(* PLC project Adressering.ecp, WAGO e!COCKPIT e!COCKPIT *)
(* stored: creationDateTime 2021-01-18T14:20:23.2110188, modificationDateTime 2021-01-18T11:51:27.6823754 *)

TYPE dtRomtype_99999999999999 : STRUCT
  RB601_V : BOOL;  (* Bevegelse *)
  RB602_V : BOOL;  (* Bevegelse *)
  RB603_V : BOOL;  (* Bevegelse *)
  RB604_V : BOOL;  (* Bevegelse *)
  RB605_V : BOOL;  (* Bevegelse *)
  RB606_V : BOOL;  (* Bevegelse *)
  RB607_V : BOOL;  (* Bevegelse *)
  RB608_V : BOOL;  (* Bevegelse *)
  RB609_V : BOOL;  (* Bevegelse *)
  RB601_HVAC : BOOL;  (* HVAC signal *)
  RB602_HVAC : BOOL;  (* HVAC signal *)
  RB603_HVAC : BOOL;  (* HVAC signal *)
  RB604_HVAC : BOOL;  (* HVAC signal *)
  RB605_HVAC : BOOL;  (* HVAC signal *)
  RB606_HVAC : BOOL;  (* HVAC signal *)
  RB607_HVAC : BOOL;  (* HVAC signal *)
  RB608_HVAC : BOOL;  (* HVAC signal *)
  RB609_HVAC : BOOL;  (* HVAC signal *)
  RT601_CT : REAL;  (* Rom temperatur *)
  RT602_CT : REAL;  (* Rom temperatur *)
  RT602_SP : REAL;  (* Temperatur SP *)
  RT603_CT : REAL;  (* Rom temperatur *)
  RT603_SP : REAL;  (* Temperatur SP *)
  RT604_CT : REAL;  (* Rom temperatur *)
  RT604_SP : REAL;  (* Temperatur SP *)
  RT605_CT : REAL;  (* Rom temperatur *)
  RT605_SP : REAL;  (* Temperatur SP *)
  RT606_CT : REAL;  (* Rom temperatur *)
  RT606_SP : REAL;  (* Temperatur SP *)
  RT607_CT : REAL;  (* Rom temperatur *)
  RT607_SP : REAL;  (* Temperatur SP *)
  RT608_CT : REAL;  (* Rom temperatur *)
  RT608_SP : REAL;  (* Temperatur SP *)
  RT609_CT : REAL;  (* Rom temperatur *)
  RT609_SP : REAL;  (* Temperatur SP *)
  RT601_SP_D : REAL;  (* Temperatur SP *)
  RT601_SP_S : REAL;  (* Temperatur SP standby *)
  RT601_SP_N : REAL;  (* Temperatur SP nattsenk *)
  RT601_SP_F : REAL;  (* Temperatur SP frostsikring *)
  RT601_CS : REAL;  (* Aktivt temperatur SP *)
  OPM : INT;  (* Rom modus *)
  OPM_CV : INT;  (* Rom modus verdi *)
  RY601_CV : REAL;  (* Co2 Nivaa *)
  RY602_CV : REAL;  (* Co2 Nivaa *)
  RY603_CV : REAL;  (* Co2 Nivaa *)
  RY604_CV : REAL;  (* Co2 Nivaa *)
  RY605_CV : REAL;  (* Co2 Nivaa *)
  RY606_CV : REAL;  (* Co2 Nivaa *)
  RY607_CV : REAL;  (* Co2 Nivaa *)
  RY608_CV : REAL;  (* Co2 Nivaa *)
  RY609_CV : REAL;  (* Co2 Nivaa *)
  RY601_SP : REAL;  (* Co2 SP *)
  RY601_OP : REAL;  (* Co2 paadrag *)
  LH601_OP : REAL;  (* Varmepaadrag *)
  LH602_OP : REAL;  (* Varmepaadrag *)
  LH603_OP : REAL;  (* Varmepaadrag *)
  LH604_OP : REAL;  (* Varmepaadrag *)
  LH605_OP : REAL;  (* Varmepaadrag *)
  LH606_OP : REAL;  (* Varmepaadrag *)
  LH607_OP : REAL;  (* Varmepaadrag *)
  LH608_OP : REAL;  (* Varmepaadrag *)
  LH609_OP : REAL;  (* Varmepaadrag *)
  LH601_MAN : BOOL;  (* Force LH *)
  LH601_CMD : BOOL;  (* LH601_CMD *)
  LH602_CMD : BOOL;  (* LH602_CMD *)
  LH603_CMD : BOOL;  (* LH603_CMD *)
  LH604_CMD : BOOL;  (* LH604_CMD *)
  LH605_CMD : BOOL;  (* LH605_CMD *)
  LH606_CMD : BOOL;  (* LH606_CMD *)
  LH607_CMD : BOOL;  (* LH607_CMD *)
  LH608_CMD : BOOL;  (* LH608_CMD *)
  LH609_CMD : BOOL;  (* LH609_CMD *)
  LC601_OP : REAL;  (* LC601_OP *)
  LC602_OP : REAL;  (* LC602_OP *)
  LC603_OP : REAL;  (* LC603_OP *)
  LC604_OP : REAL;  (* LC604_OP *)
  LC605_OP : REAL;  (* LC605_OP *)
  LC606_OP : REAL;  (* LC606_OP *)
  LC607_OP : REAL;  (* LC607_OP *)
  LC608_OP : REAL;  (* LC608_OP *)
  LC609_OP : REAL;  (* LC609_OP *)
  LC601_MAN : BOOL;  (* Force LC *)
  LC601_CMD : BOOL;  (* LC601_CMD *)
  LC602_CMD : BOOL;  (* LC602_CMD *)
  LC603_CMD : BOOL;  (* LC603_CMD *)
  LC604_CMD : BOOL;  (* LC604_CMD *)
  LC605_CMD : BOOL;  (* LC605_CMD *)
  LC606_CMD : BOOL;  (* LC606_CMD *)
  LC607_CMD : BOOL;  (* LC607_CMD *)
  LC608_CMD : BOOL;  (* LC608_CMD *)
  LC609_CMD : BOOL;  (* LC609_CMD *)
  RT601_SP : REAL;  (* Temperatur SP feedback *)
  RT601_SP_FB : REAL;  (* Temperatur SP *)
  RT601_SP_IN : REAL;  (* Temperatur SP lokalt panel *)
  RT602_SP_FB : REAL;  (* Temperatur SP *)
  RT602_SP_IN : REAL;  (* Temperatur SP lokalt panel *)
  RT603_SP_FB : REAL;  (* Temperatur SP *)
  RT603_SP_IN : REAL;  (* Temperatur SP lokalt panel *)
  RT604_SP_FB : REAL;  (* Temperatur SP *)
  RT604_SP_IN : REAL;  (* Temperatur SP lokalt panel *)
  RT605_SP_FB : REAL;  (* Temperatur SP *)
  RT605_SP_IN : REAL;  (* Temperatur SP lokalt panel *)
  RT606_SP_FB : REAL;  (* Temperatur SP *)
  RT606_SP_IN : REAL;  (* Temperatur SP lokalt panel *)
  RT607_SP_FB : REAL;  (* Temperatur SP *)
  RT607_SP_IN : REAL;  (* Temperatur SP lokalt panel *)
  RT608_SP_FB : REAL;  (* Temperatur SP *)
  RT608_SP_IN : REAL;  (* Temperatur SP lokalt panel *)
  RT609_SP_FB : REAL;  (* Temperatur SP *)
  RT609_SP_IN : REAL;  (* Temperatur SP lokalt panel *)
  LU601_V : BOOL;  (* Befukter status *)
  LU602_V : BOOL;  (* Befukter status *)
  LU603_V : BOOL;  (* Befukter status *)
  LU604_V : BOOL;  (* Befukter status *)
  LU605_V : BOOL;  (* Befukter status *)
  LU606_V : BOOL;  (* Befukter status *)
  LU607_V : BOOL;  (* Befukter status *)
  LU608_V : BOOL;  (* Befukter status *)
  LU609_V : BOOL;  (* Befukter status *)
  LU601_AL : BOOL;  (* Befukter alarm/feil *)
  LU602_AL : BOOL;  (* Befukter alarm/feil *)
  LU603_AL : BOOL;  (* Befukter alarm/feil *)
  LU604_AL : BOOL;  (* Befukter alarm/feil *)
  LU605_AL : BOOL;  (* Befukter alarm/feil *)
  LU606_AL : BOOL;  (* Befukter alarm/feil *)
  LU607_AL : BOOL;  (* Befukter alarm/feil *)
  LU608_AL : BOOL;  (* Befukter alarm/feil *)
  LU609_AL : BOOL;  (* Befukter alarm/feil *)
  LU601_CMD : BOOL;  (* Befukter tillat start *)
  LU602_CMD : BOOL;  (* Befukter tillat start *)
  LU603_CMD : BOOL;  (* Befukter tillat start *)
  LU604_CMD : BOOL;  (* Befukter tillat start *)
  LU605_CMD : BOOL;  (* Befukter tillat start *)
  LU606_CMD : BOOL;  (* Befukter tillat start *)
  LU607_CMD : BOOL;  (* Befukter tillat start *)
  LU608_CMD : BOOL;  (* Befukter tillat start *)
  LU609_CMD : BOOL;  (* Befukter tillat start *)
END_STRUCT;
END_TYPE

TYPE dtRomtype_2210111100111 : STRUCT
  RB601_V : BOOL;  (* Bevegelse *)
  RB602_V : BOOL;  (* Bevegelse *)
  RB601_HVAC : BOOL;  (* HVAC signal *)
  RB602_HVAC : BOOL;  (* HVAC signal *)
  RT601_CT : REAL;  (* Rom temperatur *)
  RT601_SP_D : REAL;  (* Temperatur SP *)
  RT601_SP_S : REAL;  (* Temperatur SP standby *)
  RT601_SP_N : REAL;  (* Temperatur SP nattsenk *)
  RT601_SP_F : REAL;  (* Temperatur SP frostsikring *)
  RT601_CS : REAL;  (* Aktivt temperatur SP *)
  OPM : INT;  (* Rom modus *)
  OPM_CV : INT;  (* Rom modus verdi *)
  LH601_OP : REAL;  (* Varmepaadrag *)
  LH601_MAN : BOOL;  (* Force LH *)
  LH601_CMD : BOOL;  (* LH601_CMD *)
  LC601_OP : REAL;  (* LC601_OP *)
  LC601_MAN : BOOL;  (* Force LC *)
  LC601_CMD : BOOL;  (* LC601_CMD *)
  LU601_V : BOOL;  (* Befukter status *)
  LU601_AL : BOOL;  (* Befukter alarm/feil *)
  LU601_CMD : BOOL;  (* Befukter tillat start *)
END_STRUCT;
END_TYPE

TYPE dtRomtype_1120011 : STRUCT
  RB601_V : BOOL;  (* Bevegelse *)
  RB601_HVAC : BOOL;  (* HVAC signal *)
  RT601_CT : REAL;  (* Rom temperatur *)
  RT602_CT : REAL;  (* Rom temperatur *)
  RT602_SP : REAL;  (* Temperatur SP *)
  RT601_SP_D : REAL;  (* Temperatur SP *)
  RT601_SP_S : REAL;  (* Temperatur SP standby *)
  RT601_SP_N : REAL;  (* Temperatur SP nattsenk *)
  RT601_SP_F : REAL;  (* Temperatur SP frostsikring *)
  RT601_CS : REAL;  (* Aktivt temperatur SP *)
  OPM : INT;  (* Rom modus *)
  OPM_CV : INT;  (* Rom modus verdi *)
  LH601_CMD : BOOL;  (* LH601_CMD *)
  LH601_MAN : BOOL;  (* Force LH *)
  LC601_OP : REAL;  (* LC601_OP *)
  LC601_MAN : BOOL;  (* Force LC *)
END_STRUCT;
END_TYPE

TYPE dtRomtype_11 : STRUCT
  RB601_V : BOOL;  (* Bevegelse *)
  RB601_HVAC : BOOL;  (* HVAC signal *)
END_STRUCT;
END_TYPE

TYPE dtRomtype_1121 : STRUCT
  RB601_V : BOOL;  (* Bevegelse *)
  RB601_HVAC : BOOL;  (* HVAC signal *)
  RT601_CT : REAL;  (* Rom temperatur *)
  RT602_CT : REAL;  (* Rom temperatur *)
  RT602_SP : REAL;  (* Temperatur SP *)
  RT601_SP_D : REAL;  (* Temperatur SP *)
  RT601_SP_S : REAL;  (* Temperatur SP standby *)
  RT601_SP_N : REAL;  (* Temperatur SP nattsenk *)
  RT601_SP_F : REAL;  (* Temperatur SP frostsikring *)
  RT601_CS : REAL;  (* Aktivt temperatur SP *)
  OPM : INT;  (* Rom modus *)
  OPM_CV : INT;  (* Rom modus verdi *)
  RY601_CV : REAL;  (* Co2 Nivaa *)
  RY601_SP : REAL;  (* Co2 SP *)
  RY601_OP : REAL;  (* Co2 paadrag *)
END_STRUCT;
END_TYPE

TYPE dtRomtype_112001 : STRUCT
  RB601_V : BOOL;  (* Bevegelse *)
  RB601_HVAC : BOOL;  (* HVAC signal *)
  RT601_CT : REAL;  (* Rom temperatur *)
  RT602_CT : REAL;  (* Rom temperatur *)
  RT602_SP : REAL;  (* Temperatur SP *)
  RT601_SP_D : REAL;  (* Temperatur SP *)
  RT601_SP_S : REAL;  (* Temperatur SP standby *)
  RT601_SP_N : REAL;  (* Temperatur SP nattsenk *)
  RT601_SP_F : REAL;  (* Temperatur SP frostsikring *)
  RT601_CS : REAL;  (* Aktivt temperatur SP *)
  OPM : INT;  (* Rom modus *)
  OPM_CV : INT;  (* Rom modus verdi *)
  LH601_CMD : BOOL;  (* LH601_CMD *)
  LH601_MAN : BOOL;  (* Force LH *)
END_STRUCT;
END_TYPE

TYPE dtRomtype_111 : STRUCT
  RB601_V : BOOL;  (* Bevegelse *)
  RB601_HVAC : BOOL;  (* HVAC signal *)
  RT601_CT : REAL;  (* Rom temperatur *)
  RT601_SP_D : REAL;  (* Temperatur SP *)
  RT601_SP_S : REAL;  (* Temperatur SP standby *)
  RT601_SP_N : REAL;  (* Temperatur SP nattsenk *)
  RT601_SP_F : REAL;  (* Temperatur SP frostsikring *)
  RT601_CS : REAL;  (* Aktivt temperatur SP *)
  OPM : INT;  (* Rom modus *)
  OPM_CV : INT;  (* Rom modus verdi *)
END_STRUCT;
END_TYPE

TYPE dtRomtype_22 : STRUCT
  RB601_V : BOOL;  (* Bevegelse *)
  RB602_V : BOOL;  (* Bevegelse *)
  RB601_HVAC : BOOL;  (* HVAC signal *)
  RB602_HVAC : BOOL;  (* HVAC signal *)
END_STRUCT;
END_TYPE

TYPE dtRomtype_4421011 : STRUCT
  RB601_V : BOOL;  (* Bevegelse *)
  RB602_V : BOOL;  (* Bevegelse *)
  RB603_V : BOOL;  (* Bevegelse *)
  RB604_V : BOOL;  (* Bevegelse *)
  RB601_HVAC : BOOL;  (* HVAC signal *)
  RB602_HVAC : BOOL;  (* HVAC signal *)
  RB603_HVAC : BOOL;  (* HVAC signal *)
  RB604_HVAC : BOOL;  (* HVAC signal *)
  RT601_CT : REAL;  (* Rom temperatur *)
  RT602_CT : REAL;  (* Rom temperatur *)
  RT602_SP : REAL;  (* Temperatur SP *)
  RT601_SP_D : REAL;  (* Temperatur SP *)
  RT601_SP_S : REAL;  (* Temperatur SP standby *)
  RT601_SP_N : REAL;  (* Temperatur SP nattsenk *)
  RT601_SP_F : REAL;  (* Temperatur SP frostsikring *)
  RT601_CS : REAL;  (* Aktivt temperatur SP *)
  OPM : INT;  (* Rom modus *)
  OPM_CV : INT;  (* Rom modus verdi *)
  RY601_CV : REAL;  (* Co2 Nivaa *)
  RY601_SP : REAL;  (* Co2 SP *)
  RY601_OP : REAL;  (* Co2 paadrag *)
  LH601_CMD : BOOL;  (* LH601_CMD *)
  LH601_MAN : BOOL;  (* Force LH *)
  LC601_OP : REAL;  (* LC601_OP *)
  LC601_MAN : BOOL;  (* Force LC *)
END_STRUCT;
END_TYPE

TYPE dtRomtype_003 : STRUCT
  RT601_CT : REAL;  (* Rom temperatur *)
  RT602_CT : REAL;  (* Rom temperatur *)
  RT602_SP : REAL;  (* Temperatur SP *)
  RT603_CT : REAL;  (* Rom temperatur *)
  RT603_SP : REAL;  (* Temperatur SP *)
  RT601_SP_D : REAL;  (* Temperatur SP *)
  RT601_SP_S : REAL;  (* Temperatur SP standby *)
  RT601_SP_N : REAL;  (* Temperatur SP nattsenk *)
  RT601_SP_F : REAL;  (* Temperatur SP frostsikring *)
  RT601_CS : REAL;  (* Aktivt temperatur SP *)
  OPM : INT;  (* Rom modus *)
  OPM_CV : INT;  (* Rom modus verdi *)
END_STRUCT;
END_TYPE

TYPE dtRomtype_1121011 : STRUCT
  RB601_V : BOOL;  (* Bevegelse *)
  RB601_HVAC : BOOL;  (* HVAC signal *)
  RT601_CT : REAL;  (* Rom temperatur *)
  RT602_CT : REAL;  (* Rom temperatur *)
  RT602_SP : REAL;  (* Temperatur SP *)
  RT601_SP_D : REAL;  (* Temperatur SP *)
  RT601_SP_S : REAL;  (* Temperatur SP standby *)
  RT601_SP_N : REAL;  (* Temperatur SP nattsenk *)
  RT601_SP_F : REAL;  (* Temperatur SP frostsikring *)
  RT601_CS : REAL;  (* Aktivt temperatur SP *)
  OPM : INT;  (* Rom modus *)
  OPM_CV : INT;  (* Rom modus verdi *)
  RY601_CV : REAL;  (* Co2 Nivaa *)
  RY601_SP : REAL;  (* Co2 SP *)
  RY601_OP : REAL;  (* Co2 paadrag *)
  LH601_CMD : BOOL;  (* LH601_CMD *)
  LH601_MAN : BOOL;  (* Force LH *)
  LC601_OP : REAL;  (* LC601_OP *)
  LC601_MAN : BOOL;  (* Force LC *)
END_STRUCT;
END_TYPE

TYPE dtRomtype_112 : STRUCT
  RB601_V : BOOL;  (* Bevegelse *)
  RB601_HVAC : BOOL;  (* HVAC signal *)
  RT601_CT : REAL;  (* Rom temperatur *)
  RT602_CT : REAL;  (* Rom temperatur *)
  RT602_SP : REAL;  (* Temperatur SP *)
  RT601_SP_D : REAL;  (* Temperatur SP *)
  RT601_SP_S : REAL;  (* Temperatur SP standby *)
  RT601_SP_N : REAL;  (* Temperatur SP nattsenk *)
  RT601_SP_F : REAL;  (* Temperatur SP frostsikring *)
  RT601_CS : REAL;  (* Aktivt temperatur SP *)
  OPM : INT;  (* Rom modus *)
  OPM_CV : INT;  (* Rom modus verdi *)
END_STRUCT;
END_TYPE

{attribute 'qualified_only'}
VAR_GLOBAL  (* STLV59_563 *)
  STLV59_A_563_KNX_Card_1_Status : BOOL;  (* KNX kort 1 status *)
  STLV59_A_563_000 : dtRomtype_99999999999999;
  STLV59_A_563_001 : dtRomtype_2210111100111;
  STLV59_A_563_002 : dtRomtype_1120011;
  STLV59_A_563_003 : dtRomtype_11;
  STLV59_A_563_004 : dtRomtype_1121;
  STLV59_A_563_005 : dtRomtype_112001;
  STLV59_A_563_006 : dtRomtype_111;
  STLV59_A_563_007 : dtRomtype_112001;
  STLV59_A_563_008 : dtRomtype_112001;
  STLV59_A_563_009 : dtRomtype_112001;
  STLV59_A_563_010 : dtRomtype_112001;
  STLV59_A_563_011 : dtRomtype_112001;
  STLV59_A_563_012 : dtRomtype_112001;
  STLV59_A_563_013 : dtRomtype_112001;
  STLV59_A_563_014 : dtRomtype_22;
  STLV59_A_563_015 : dtRomtype_11;
  STLV59_A_563_016 : dtRomtype_11;
  STLV59_A_563_017 : dtRomtype_112001;
  STLV59_A_563_101 : dtRomtype_112001;
  STLV59_A_563_102 : dtRomtype_112001;
  STLV59_A_563_103 : dtRomtype_4421011;
  STLV59_A_563_109 : dtRomtype_112001;
  STLV59_A_563_201 : dtRomtype_003;
  STLV59_A_563_212 : dtRomtype_1121011;
  STLV59_A_563_213 : dtRomtype_112;
  STLV59_A_563_T2_1 : dtRomtype_112001;
  STLV59_A_563_T2_2 : dtRomtype_112001;
END_VAR

FUNCTION_BLOCK fbRomtype_99999999999999
  VAR_INPUT
    RB601_HVAC : BOOL;
    RB602_HVAC : BOOL;
    RB603_HVAC : BOOL;
    RB604_HVAC : BOOL;
    RB605_HVAC : BOOL;
    RB606_HVAC : BOOL;
    RB607_HVAC : BOOL;
    RB608_HVAC : BOOL;
    RB609_HVAC : BOOL;
    RT601_CT : REAL;
    RT602_CT : REAL;
    RT602_SP : REAL;
    RT603_CT : REAL;
    RT603_SP : REAL;
    RT604_CT : REAL;
    RT604_SP : REAL;
    RT605_CT : REAL;
    RT605_SP : REAL;
    RT606_CT : REAL;
    RT606_SP : REAL;
    RT607_CT : REAL;
    RT607_SP : REAL;
    RT608_CT : REAL;
    RT608_SP : REAL;
    RT609_CT : REAL;
    RT609_SP : REAL;
    RT601_SP_D : REAL;
    RT601_SP_S : REAL;
    RT601_SP_N : REAL;
    RT601_SP_F : REAL;
    OPM : INT;
    RY601_CV : REAL;
    RY602_CV : REAL;
    RY603_CV : REAL;
    RY604_CV : REAL;
    RY605_CV : REAL;
    RY606_CV : REAL;
    RY607_CV : REAL;
    RY608_CV : REAL;
    RY609_CV : REAL;
    RY601_SP : REAL;
    LH601_MAN : BOOL;
    LC601_MAN : BOOL;
    RT601_SP_IN : REAL;
    RT602_SP_IN : REAL;
    RT603_SP_IN : REAL;
    RT604_SP_IN : REAL;
    RT605_SP_IN : REAL;
    RT606_SP_IN : REAL;
    RT607_SP_IN : REAL;
    RT608_SP_IN : REAL;
    RT609_SP_IN : REAL;
    LU601_V : BOOL;
    LU602_V : BOOL;
    LU603_V : BOOL;
    LU604_V : BOOL;
    LU605_V : BOOL;
    LU606_V : BOOL;
    LU607_V : BOOL;
    LU608_V : BOOL;
    LU609_V : BOOL;
    LU601_AL : BOOL;
    LU602_AL : BOOL;
    LU603_AL : BOOL;
    LU604_AL : BOOL;
    LU605_AL : BOOL;
    LU606_AL : BOOL;
    LU607_AL : BOOL;
    LU608_AL : BOOL;
    LU609_AL : BOOL;
  END_VAR
  VAR_OUTPUT
    OPM_CV : INT;
    RT601_CS : REAL;
    RT602_CS : REAL;
    RT603_CS : REAL;
    RT604_CS : REAL;
    RT605_CS : REAL;
    RT606_CS : REAL;
    RT607_CS : REAL;
    RT608_CS : REAL;
    RT609_CS : REAL;
    RY601_OP : REAL;
    LH601_OP : REAL;
    LH602_OP : REAL;
    LH603_OP : REAL;
    LH604_OP : REAL;
    LH605_OP : REAL;
    LH606_OP : REAL;
    LH607_OP : REAL;
    LH608_OP : REAL;
    LH609_OP : REAL;
    LH601_CMD : BOOL;
    LH602_CMD : BOOL;
    LH603_CMD : BOOL;
    LH604_CMD : BOOL;
    LH605_CMD : BOOL;
    LH606_CMD : BOOL;
    LH607_CMD : BOOL;
    LH608_CMD : BOOL;
    LH609_CMD : BOOL;
    LC601_OP : REAL;
    LC602_OP : REAL;
    LC603_OP : REAL;
    LC604_OP : REAL;
    LC605_OP : REAL;
    LC606_OP : REAL;
    LC607_OP : REAL;
    LC608_OP : REAL;
    LC609_OP : REAL;
    LC601_CMD : BOOL;
    LC602_CMD : BOOL;
    LC603_CMD : BOOL;
    LC604_CMD : BOOL;
    LC605_CMD : BOOL;
    LC606_CMD : BOOL;
    LC607_CMD : BOOL;
    LC608_CMD : BOOL;
    LC609_CMD : BOOL;
    LU601_CMD : BOOL;
    LU602_CMD : BOOL;
    LU603_CMD : BOOL;
    LU604_CMD : BOOL;
    LU605_CMD : BOOL;
    LU606_CMD : BOOL;
    LU607_CMD : BOOL;
    LU608_CMD : BOOL;
    LU609_CMD : BOOL;
  END_VAR

(* CFC diagram, written out as Structured Text *)
END_FUNCTION_BLOCK

FUNCTION_BLOCK fbRomtype_2210111100111
  VAR_INPUT
    RB601_HVAC : BOOL;
    RB602_HVAC : BOOL;
    RT601_CT : REAL;
    RT601_SP_D : REAL;
    RT601_SP_S : REAL;
    RT601_SP_N : REAL;
    RT601_SP_F : REAL;
    OPM : INT;
    LH601_MAN : BOOL;
    LC601_MAN : BOOL;
    LU601_V : BOOL;
    LU601_AL : BOOL;
  END_VAR
  VAR_OUTPUT
    OPM_CV : INT;
    RT601_CS : REAL;
    LH601_OP : REAL;
    LH601_CMD : BOOL;
    LC601_OP : REAL;
    LC601_CMD : BOOL;
    LU601_CMD : BOOL;
  END_VAR

(* CFC diagram, written out as Structured Text *)
END_FUNCTION_BLOCK

FUNCTION_BLOCK fbRomtype_1120011
  VAR_INPUT
    RB601_HVAC : BOOL;
    RT601_CT : REAL;
    RT602_CT : REAL;
    RT602_SP : REAL;
    RT601_SP_D : REAL;
    RT601_SP_S : REAL;
    RT601_SP_N : REAL;
    RT601_SP_F : REAL;
    OPM : INT;
    LH601_MAN : BOOL;
    LC601_MAN : BOOL;
  END_VAR
  VAR_OUTPUT
    OPM_CV : INT;
    RT601_CS : REAL;
    RT602_CS : REAL;
    LH601_CMD : BOOL;
    LC601_OP : REAL;
  END_VAR

(* CFC diagram, written out as Structured Text *)
END_FUNCTION_BLOCK

FUNCTION_BLOCK fbRomtype_1121
  VAR_INPUT
    RB601_HVAC : BOOL;
    RT601_CT : REAL;
    RT602_CT : REAL;
    RT602_SP : REAL;
    RT601_SP_D : REAL;
    RT601_SP_S : REAL;
    RT601_SP_N : REAL;
    RT601_SP_F : REAL;
    OPM : INT;
    RY601_CV : REAL;
    RY601_SP : REAL;
  END_VAR
  VAR_OUTPUT
    OPM_CV : INT;
    RT601_CS : REAL;
    RT602_CS : REAL;
    RY601_OP : REAL;
  END_VAR

(* CFC diagram, written out as Structured Text *)
END_FUNCTION_BLOCK

FUNCTION_BLOCK fbRomtype_112001
  VAR_INPUT
    RB601_HVAC : BOOL;
    RT601_CT : REAL;
    RT602_CT : REAL;
    RT602_SP : REAL;
    RT601_SP_D : REAL;
    RT601_SP_S : REAL;
    RT601_SP_N : REAL;
    RT601_SP_F : REAL;
    OPM : INT;
    LH601_MAN : BOOL;
  END_VAR
  VAR_OUTPUT
    OPM_CV : INT;
    RT601_CS : REAL;
    RT602_CS : REAL;
    LH601_CMD : BOOL;
  END_VAR

(* CFC diagram, written out as Structured Text *)
END_FUNCTION_BLOCK

FUNCTION_BLOCK fbRomtype_4421011
  VAR_INPUT
    RB601_HVAC : BOOL;
    RB602_HVAC : BOOL;
    RB603_HVAC : BOOL;
    RB604_HVAC : BOOL;
    RT601_CT : REAL;
    RT602_CT : REAL;
    RT602_SP : REAL;
    RT601_SP_D : REAL;
    RT601_SP_S : REAL;
    RT601_SP_N : REAL;
    RT601_SP_F : REAL;
    OPM : INT;
    RY601_CV : REAL;
    RY601_SP : REAL;
    LH601_MAN : BOOL;
    LC601_MAN : BOOL;
  END_VAR
  VAR_OUTPUT
    OPM_CV : INT;
    RT601_CS : REAL;
    RT602_CS : REAL;
    RY601_OP : REAL;
    LH601_CMD : BOOL;
    LC601_OP : REAL;
  END_VAR

(* CFC diagram, written out as Structured Text *)
END_FUNCTION_BLOCK

FUNCTION_BLOCK fbRomtype_1121011
  VAR_INPUT
    RB601_HVAC : BOOL;
    RT601_CT : REAL;
    RT602_CT : REAL;
    RT602_SP : REAL;
    RT601_SP_D : REAL;
    RT601_SP_S : REAL;
    RT601_SP_N : REAL;
    RT601_SP_F : REAL;
    OPM : INT;
    RY601_CV : REAL;
    RY601_SP : REAL;
    LH601_MAN : BOOL;
    LC601_MAN : BOOL;
  END_VAR
  VAR_OUTPUT
    OPM_CV : INT;
    RT601_CS : REAL;
    RT602_CS : REAL;
    RY601_OP : REAL;
    LH601_CMD : BOOL;
    LC601_OP : REAL;
  END_VAR

(* CFC diagram, written out as Structured Text *)
END_FUNCTION_BLOCK

PROGRAM PRG_563_KNX_1
  VAR
    i : INT := 0;  (* Felles *)
    Interval : OSCAT_BASIC.CLK_PRG;
    typDPT : typDPT;
    KNX_master_1 : WagoAppKNX.FbKNX_Master;  (* Master *)
    M1_001_000_RB601_V : fbDPT_Switch_pro;  (* 000 *)
    M1_002_000_RB602_V : fbDPT_Switch_pro;
    M1_003_000_RB603_V : fbDPT_Switch_pro;
    M1_004_000_RB604_V : fbDPT_Switch_pro;
    M1_005_000_RB605_V : fbDPT_Switch_pro;
    M1_006_000_RB606_V : fbDPT_Switch_pro;
    M1_007_000_RB607_V : fbDPT_Switch_pro;
    M1_008_000_RB608_V : fbDPT_Switch_pro;
    M1_009_000_RB609_V : fbDPT_Switch_pro;
    M1_010_000_RB601_HVAC : fbDPT_Switch_pro;
    M1_011_000_RB602_HVAC : fbDPT_Switch_pro;
    M1_012_000_RB603_HVAC : fbDPT_Switch_pro;
    M1_013_000_RB604_HVAC : fbDPT_Switch_pro;
    M1_014_000_RB605_HVAC : fbDPT_Switch_pro;
    M1_015_000_RB606_HVAC : fbDPT_Switch_pro;
    M1_016_000_RB607_HVAC : fbDPT_Switch_pro;
    M1_017_000_RB608_HVAC : fbDPT_Switch_pro;
    M1_018_000_RB609_HVAC : fbDPT_Switch_pro;
    M1_019_000_RT601_CT : fbDPT_Value_Temp_pro;
    M1_020_000_RT602_CT : fbDPT_Value_Temp_pro;
    M1_021_000_RT603_CT : fbDPT_Value_Temp_pro;
    M1_022_000_RT604_CT : fbDPT_Value_Temp_pro;
    M1_023_000_RT605_CT : fbDPT_Value_Temp_pro;
    M1_024_000_RT606_CT : fbDPT_Value_Temp_pro;
    M1_025_000_RT607_CT : fbDPT_Value_Temp_pro;
    M1_026_000_RT608_CT : fbDPT_Value_Temp_pro;
    M1_027_000_RT609_CT : fbDPT_Value_Temp_pro;
    M1_028_000_RY601_CV : fbDPT_Value_AirQuality_pro;
    M1_029_000_RY602_CV : fbDPT_Value_AirQuality_pro;
    M1_030_000_RY603_CV : fbDPT_Value_AirQuality_pro;
    M1_031_000_RY604_CV : fbDPT_Value_AirQuality_pro;
    M1_032_000_RY605_CV : fbDPT_Value_AirQuality_pro;
    M1_033_000_RY606_CV : fbDPT_Value_AirQuality_pro;
    M1_034_000_RY607_CV : fbDPT_Value_AirQuality_pro;
    M1_035_000_RY608_CV : fbDPT_Value_AirQuality_pro;
    M1_036_000_RY609_CV : fbDPT_Value_AirQuality_pro;
    M1_037_000_LH601_OP : fbDPT_Scaling_pro;
    M1_038_000_LH602_OP : fbDPT_Scaling_pro;
    M1_039_000_LH603_OP : fbDPT_Scaling_pro;
    M1_040_000_LH604_OP : fbDPT_Scaling_pro;
    M1_041_000_LH605_OP : fbDPT_Scaling_pro;
    M1_042_000_LH606_OP : fbDPT_Scaling_pro;
    M1_043_000_LH607_OP : fbDPT_Scaling_pro;
    M1_044_000_LH608_OP : fbDPT_Scaling_pro;
    M1_045_000_LH609_OP : fbDPT_Scaling_pro;
    M1_046_000_LH601_CMD : fbDPT_Switch_pro;
    M1_047_000_LH602_CMD : fbDPT_Switch_pro;
    M1_048_000_LH603_CMD : fbDPT_Switch_pro;
    M1_049_000_LH604_CMD : fbDPT_Switch_pro;
    M1_050_000_LH605_CMD : fbDPT_Switch_pro;
    M1_051_000_LH606_CMD : fbDPT_Switch_pro;
    M1_052_000_LH607_CMD : fbDPT_Switch_pro;
    M1_053_000_LH608_CMD : fbDPT_Switch_pro;
    M1_054_000_LH609_CMD : fbDPT_Switch_pro;
    M1_055_000_LC601_OP : fbDPT_Scaling_pro;
    M1_056_000_LC602_OP : fbDPT_Scaling_pro;
    M1_057_000_LC603_OP : fbDPT_Scaling_pro;
    M1_058_000_LC604_OP : fbDPT_Scaling_pro;
    M1_059_000_LC605_OP : fbDPT_Scaling_pro;
    M1_060_000_LC606_OP : fbDPT_Scaling_pro;
    M1_061_000_LC607_OP : fbDPT_Scaling_pro;
    M1_062_000_LC608_OP : fbDPT_Scaling_pro;
    M1_063_000_LC609_OP : fbDPT_Scaling_pro;
    M1_064_000_LC601_CMD : fbDPT_Switch_pro;
    M1_065_000_LC602_CMD : fbDPT_Switch_pro;
    M1_066_000_LC603_CMD : fbDPT_Switch_pro;
    M1_067_000_LC604_CMD : fbDPT_Switch_pro;
    M1_068_000_LC605_CMD : fbDPT_Switch_pro;
    M1_069_000_LC606_CMD : fbDPT_Switch_pro;
    M1_070_000_LC607_CMD : fbDPT_Switch_pro;
    M1_071_000_LC608_CMD : fbDPT_Switch_pro;
    M1_072_000_LC609_CMD : fbDPT_Switch_pro;
    M1_073_000_RT601_SP : fbDPT_Value_Temp_pro;
    M1_074_000_RT602_SP : fbDPT_Value_Temp_pro;
    M1_075_000_RT603_SP : fbDPT_Value_Temp_pro;
    M1_076_000_RT604_SP : fbDPT_Value_Temp_pro;
    M1_077_000_RT605_SP : fbDPT_Value_Temp_pro;
    M1_078_000_RT606_SP : fbDPT_Value_Temp_pro;
    M1_079_000_RT607_SP : fbDPT_Value_Temp_pro;
    M1_080_000_RT608_SP : fbDPT_Value_Temp_pro;
    M1_081_000_RT609_SP : fbDPT_Value_Temp_pro;
    M1_082_000_RT601_SP_FB : fbDPT_Value_Temp_pro;
    M1_083_000_RT602_SP_FB : fbDPT_Value_Temp_pro;
    M1_084_000_RT603_SP_FB : fbDPT_Value_Temp_pro;
    M1_085_000_RT604_SP_FB : fbDPT_Value_Temp_pro;
    M1_086_000_RT605_SP_FB : fbDPT_Value_Temp_pro;
    M1_087_000_RT606_SP_FB : fbDPT_Value_Temp_pro;
    M1_088_000_RT607_SP_FB : fbDPT_Value_Temp_pro;
    M1_089_000_RT608_SP_FB : fbDPT_Value_Temp_pro;
    M1_090_000_RT609_SP_FB : fbDPT_Value_Temp_pro;
    M1_091_000_LU601_V : fbDPT_Switch_pro;
    M1_092_000_LU602_V : fbDPT_Switch_pro;
    M1_093_000_LU603_V : fbDPT_Switch_pro;
    M1_094_000_LU604_V : fbDPT_Switch_pro;
    M1_095_000_LU605_V : fbDPT_Switch_pro;
    M1_096_000_LU606_V : fbDPT_Switch_pro;
    M1_097_000_LU607_V : fbDPT_Switch_pro;
    M1_098_000_LU608_V : fbDPT_Switch_pro;
    M1_099_000_LU609_V : fbDPT_Switch_pro;
    M1_100_000_LU601_AL : fbDPT_Switch_pro;
    M1_101_000_LU602_AL : fbDPT_Switch_pro;
    M1_102_000_LU603_AL : fbDPT_Switch_pro;
    M1_103_000_LU604_AL : fbDPT_Switch_pro;
    M1_104_000_LU605_AL : fbDPT_Switch_pro;
    M1_105_000_LU606_AL : fbDPT_Switch_pro;
    M1_106_000_LU607_AL : fbDPT_Switch_pro;
    M1_107_000_LU608_AL : fbDPT_Switch_pro;
    M1_108_000_LU609_AL : fbDPT_Switch_pro;
    M1_109_000_LU601_CMD : fbDPT_Switch_pro;
    M1_110_000_LU602_CMD : fbDPT_Switch_pro;
    M1_111_000_LU603_CMD : fbDPT_Switch_pro;
    M1_112_000_LU604_CMD : fbDPT_Switch_pro;
    M1_113_000_LU605_CMD : fbDPT_Switch_pro;
    M1_114_000_LU606_CMD : fbDPT_Switch_pro;
    M1_115_000_LU607_CMD : fbDPT_Switch_pro;
    M1_116_000_LU608_CMD : fbDPT_Switch_pro;
    M1_117_000_LU609_CMD : fbDPT_Switch_pro;
    M1_118_001_RB601_V : fbDPT_Switch_pro;  (* 001 *)
    M1_119_001_RB602_V : fbDPT_Switch_pro;
    M1_120_001_RB601_HVAC : fbDPT_Switch_pro;
    M1_121_001_RB602_HVAC : fbDPT_Switch_pro;
    M1_122_001_RT601_CT : fbDPT_Value_Temp_pro;
    M1_123_001_LH601_OP : fbDPT_Scaling_pro;
    M1_124_001_LH601_CMD : fbDPT_Switch_pro;
    M1_125_001_LC601_OP : fbDPT_Scaling_pro;
    M1_126_001_LC601_CMD : fbDPT_Switch_pro;
    M1_127_001_LU601_V : fbDPT_Switch_pro;
    M1_128_001_LU601_AL : fbDPT_Switch_pro;
    M1_129_001_LU601_CMD : fbDPT_Switch_pro;
    M1_130_002_RB601_V : fbDPT_Switch_pro;  (* 002 *)
    M1_131_002_RB601_HVAC : fbDPT_Switch_pro;
    M1_132_002_RT601_CT : fbDPT_Value_Temp_pro;
    M1_133_002_RT602_CT : fbDPT_Value_Temp_pro;
    M1_134_003_RB601_V : fbDPT_Switch_pro;  (* 003 *)
    M1_135_003_RB601_HVAC : fbDPT_Switch_pro;
    M1_136_004_RB601_V : fbDPT_Switch_pro;  (* 004 *)
    M1_137_004_RB601_HVAC : fbDPT_Switch_pro;
    M1_138_004_RT601_CT : fbDPT_Value_Temp_pro;
    M1_139_004_RT602_CT : fbDPT_Value_Temp_pro;
    M1_140_004_RY601_CV : fbDPT_Value_AirQuality_pro;
    M1_141_005_RB601_V : fbDPT_Switch_pro;  (* 005 *)
    M1_142_005_RB601_HVAC : fbDPT_Switch_pro;
    M1_143_005_RT601_CT : fbDPT_Value_Temp_pro;
    M1_144_005_RT602_CT : fbDPT_Value_Temp_pro;
    M1_145_006_RB601_V : fbDPT_Switch_pro;  (* 006 *)
    M1_146_006_RB601_HVAC : fbDPT_Switch_pro;
    M1_147_006_RT601_CT : fbDPT_Value_Temp_pro;
    M1_148_007_RB601_V : fbDPT_Switch_pro;  (* 007 *)
    M1_149_007_RB601_HVAC : fbDPT_Switch_pro;
    M1_150_007_RT601_CT : fbDPT_Value_Temp_pro;
    M1_151_007_RT602_CT : fbDPT_Value_Temp_pro;
    M1_152_008_RB601_V : fbDPT_Switch_pro;  (* 008 *)
    M1_153_008_RB601_HVAC : fbDPT_Switch_pro;
    M1_154_008_RT601_CT : fbDPT_Value_Temp_pro;
    M1_155_008_RT602_CT : fbDPT_Value_Temp_pro;
    M1_156_009_RB601_V : fbDPT_Switch_pro;  (* 009 *)
    M1_157_009_RB601_HVAC : fbDPT_Switch_pro;
    M1_158_009_RT601_CT : fbDPT_Value_Temp_pro;
    M1_159_009_RT602_CT : fbDPT_Value_Temp_pro;
    M1_160_010_RB601_V : fbDPT_Switch_pro;  (* 010 *)
    M1_161_010_RB601_HVAC : fbDPT_Switch_pro;
    M1_162_010_RT601_CT : fbDPT_Value_Temp_pro;
    M1_163_010_RT602_CT : fbDPT_Value_Temp_pro;
    M1_164_011_RB601_V : fbDPT_Switch_pro;  (* 011 *)
    M1_165_011_RB601_HVAC : fbDPT_Switch_pro;
    M1_166_011_RT601_CT : fbDPT_Value_Temp_pro;
    M1_167_011_RT602_CT : fbDPT_Value_Temp_pro;
    M1_168_012_RB601_V : fbDPT_Switch_pro;  (* 012 *)
    M1_169_012_RB601_HVAC : fbDPT_Switch_pro;
    M1_170_012_RT601_CT : fbDPT_Value_Temp_pro;
    M1_171_012_RT602_CT : fbDPT_Value_Temp_pro;
    M1_172_013_RB601_V : fbDPT_Switch_pro;  (* 013 *)
    M1_173_013_RB601_HVAC : fbDPT_Switch_pro;
    M1_174_013_RT601_CT : fbDPT_Value_Temp_pro;
    M1_175_013_RT602_CT : fbDPT_Value_Temp_pro;
    M1_176_014_RB601_V : fbDPT_Switch_pro;  (* 014 *)
    M1_177_014_RB602_V : fbDPT_Switch_pro;
    M1_178_014_RB601_HVAC : fbDPT_Switch_pro;
    M1_179_014_RB602_HVAC : fbDPT_Switch_pro;
    M1_180_015_RB601_V : fbDPT_Switch_pro;  (* 015 *)
    M1_181_015_RB601_HVAC : fbDPT_Switch_pro;
    M1_182_016_RB601_V : fbDPT_Switch_pro;  (* 016 *)
    M1_183_016_RB601_HVAC : fbDPT_Switch_pro;
    M1_184_017_RB601_V : fbDPT_Switch_pro;  (* 017 *)
    M1_185_017_RB601_HVAC : fbDPT_Switch_pro;
    M1_186_017_RT601_CT : fbDPT_Value_Temp_pro;
    M1_187_017_RT602_CT : fbDPT_Value_Temp_pro;
    M1_188_101_RB601_V : fbDPT_Switch_pro;  (* 101 *)
    M1_189_101_RB601_HVAC : fbDPT_Switch_pro;
    M1_190_101_RT601_CT : fbDPT_Value_Temp_pro;
    M1_191_101_RT602_CT : fbDPT_Value_Temp_pro;
    M1_192_102_RB601_V : fbDPT_Switch_pro;  (* 102 *)
    M1_193_102_RB601_HVAC : fbDPT_Switch_pro;
    M1_194_102_RT601_CT : fbDPT_Value_Temp_pro;
    M1_195_102_RT602_CT : fbDPT_Value_Temp_pro;
    M1_196_103_RB601_V : fbDPT_Switch_pro;  (* 103 *)
    M1_197_103_RB602_V : fbDPT_Switch_pro;
    M1_198_103_RB603_V : fbDPT_Switch_pro;
    M1_199_103_RB604_V : fbDPT_Switch_pro;
    M1_200_103_RB601_HVAC : fbDPT_Switch_pro;
    M1_201_103_RB602_HVAC : fbDPT_Switch_pro;
    M1_202_103_RB603_HVAC : fbDPT_Switch_pro;
    M1_203_103_RB604_HVAC : fbDPT_Switch_pro;
    M1_204_103_RT601_CT : fbDPT_Value_Temp_pro;
    M1_205_103_RT602_CT : fbDPT_Value_Temp_pro;
    M1_206_103_RY601_CV : fbDPT_Value_AirQuality_pro;
    M1_207_109_RB601_V : fbDPT_Switch_pro;  (* 109 *)
    M1_208_109_RB601_HVAC : fbDPT_Switch_pro;
    M1_209_109_RT601_CT : fbDPT_Value_Temp_pro;
    M1_210_109_RT602_CT : fbDPT_Value_Temp_pro;
    M1_211_201_RT601_CT : fbDPT_Value_Temp_pro;  (* 201 *)
    M1_212_201_RT602_CT : fbDPT_Value_Temp_pro;
    M1_213_201_RT603_CT : fbDPT_Value_Temp_pro;
    M1_214_212_RB601_V : fbDPT_Switch_pro;  (* 212 *)
    M1_215_212_RB601_HVAC : fbDPT_Switch_pro;
    M1_216_212_RT601_CT : fbDPT_Value_Temp_pro;
    M1_217_212_RT602_CT : fbDPT_Value_Temp_pro;
    M1_218_212_RY601_CV : fbDPT_Value_AirQuality_pro;
    M1_219_213_RB601_V : fbDPT_Switch_pro;  (* 213 *)
    M1_220_213_RB601_HVAC : fbDPT_Switch_pro;
    M1_221_213_RT601_CT : fbDPT_Value_Temp_pro;
    M1_222_213_RT602_CT : fbDPT_Value_Temp_pro;
    M1_223_T2_1_RB601_V : fbDPT_Switch_pro;  (* T2_1 *)
    M1_224_T2_1_RB601_HVAC : fbDPT_Switch_pro;
    M1_225_T2_1_RT601_CT : fbDPT_Value_Temp_pro;
    M1_226_T2_1_RT602_CT : fbDPT_Value_Temp_pro;
    M1_227_T2_2_RB601_V : fbDPT_Switch_pro;  (* T2_2 *)
    M1_228_T2_2_RB601_HVAC : fbDPT_Switch_pro;
    M1_229_T2_2_RT601_CT : fbDPT_Value_Temp_pro;
    M1_230_T2_2_RT602_CT : fbDPT_Value_Temp_pro;
  END_VAR
  VAR  (* added by the conversion: wires and edge detectors of the diagram *)
    _ADD9_OUT : INT;
    _GT15_OUT : BOOL;
    _MOVE19_ENO : BOOL;
    _MOVE19_OUT : INT;
  END_VAR

(* CFC diagram, written out as Structured Text *)
(* KNX Sending interval *)
(* KNX Master *)
Interval(PT := t#2M);
_ADD9_OUT := BOOL_TO_INT(Interval.Q) + i;
i := _ADD9_OUT;
_GT15_OUT := i > 9;
_MOVE19_OUT := MOVE(EN := _GT15_OUT, IN := 0, ENO => _MOVE19_ENO);
IF _MOVE19_ENO THEN i := _MOVE19_OUT; END_IF;
KNX_master_1(I_Port := IoConfig_Globals.KNX_EIB_TP1_Interface, bPortKNX := 1);
STLV59_563.STLV59_A_563_KNX_Card_1_Status := KNX_master_1.sStatus = 'OK';
(* Rom 000 *)
(* RB601_V *)
(* RB602_V *)
M1_001_000_RB601_V(bPortKNX := 1, dwIndex_DPT := 1, typDPT := typDPT);
STLV59_563.STLV59_A_563_000.RB601_V := M1_001_000_RB601_V.xSwitch_OUT;
M1_002_000_RB602_V(bPortKNX := 1, dwIndex_DPT := 2, typDPT := typDPT);
STLV59_563.STLV59_A_563_000.RB602_V := M1_002_000_RB602_V.xSwitch_OUT;
(* RB603_V *)
(* RB604_V *)
M1_003_000_RB603_V(bPortKNX := 1, dwIndex_DPT := 3, typDPT := typDPT);
STLV59_563.STLV59_A_563_000.RB603_V := M1_003_000_RB603_V.xSwitch_OUT;
M1_004_000_RB604_V(bPortKNX := 1, dwIndex_DPT := 4, typDPT := typDPT);
STLV59_563.STLV59_A_563_000.RB604_V := M1_004_000_RB604_V.xSwitch_OUT;
(* RB605_V *)
(* RB606_V *)
M1_005_000_RB605_V(bPortKNX := 1, dwIndex_DPT := 5, typDPT := typDPT);
STLV59_563.STLV59_A_563_000.RB605_V := M1_005_000_RB605_V.xSwitch_OUT;
M1_006_000_RB606_V(bPortKNX := 1, dwIndex_DPT := 6, typDPT := typDPT);
STLV59_563.STLV59_A_563_000.RB606_V := M1_006_000_RB606_V.xSwitch_OUT;
(* RB607_V *)
(* RB608_V *)
M1_007_000_RB607_V(bPortKNX := 1, dwIndex_DPT := 7, typDPT := typDPT);
STLV59_563.STLV59_A_563_000.RB607_V := M1_007_000_RB607_V.xSwitch_OUT;
M1_008_000_RB608_V(bPortKNX := 1, dwIndex_DPT := 8, typDPT := typDPT);
STLV59_563.STLV59_A_563_000.RB608_V := M1_008_000_RB608_V.xSwitch_OUT;
(* RB609_V *)
(* RB601_HVAC *)
M1_009_000_RB609_V(bPortKNX := 1, dwIndex_DPT := 9, typDPT := typDPT);
STLV59_563.STLV59_A_563_000.RB609_V := M1_009_000_RB609_V.xSwitch_OUT;
M1_010_000_RB601_HVAC(bPortKNX := 1, dwIndex_DPT := 10, typDPT := typDPT);
STLV59_563.STLV59_A_563_000.RB601_HVAC := M1_010_000_RB601_HVAC.xSwitch_OUT;
(* RB602_HVAC *)
(* RB603_HVAC *)
M1_011_000_RB602_HVAC(bPortKNX := 1, dwIndex_DPT := 11, typDPT := typDPT);
STLV59_563.STLV59_A_563_000.RB602_HVAC := M1_011_000_RB602_HVAC.xSwitch_OUT;
M1_012_000_RB603_HVAC(bPortKNX := 1, dwIndex_DPT := 12, typDPT := typDPT);
STLV59_563.STLV59_A_563_000.RB603_HVAC := M1_012_000_RB603_HVAC.xSwitch_OUT;
(* RB604_HVAC *)
(* RB605_HVAC *)
M1_013_000_RB604_HVAC(bPortKNX := 1, dwIndex_DPT := 13, typDPT := typDPT);
STLV59_563.STLV59_A_563_000.RB604_HVAC := M1_013_000_RB604_HVAC.xSwitch_OUT;
M1_014_000_RB605_HVAC(bPortKNX := 1, dwIndex_DPT := 14, typDPT := typDPT);
STLV59_563.STLV59_A_563_000.RB605_HVAC := M1_014_000_RB605_HVAC.xSwitch_OUT;
(* RB606_HVAC *)
(* RB607_HVAC *)
M1_015_000_RB606_HVAC(bPortKNX := 1, dwIndex_DPT := 15, typDPT := typDPT);
STLV59_563.STLV59_A_563_000.RB606_HVAC := M1_015_000_RB606_HVAC.xSwitch_OUT;
M1_016_000_RB607_HVAC(bPortKNX := 1, dwIndex_DPT := 16, typDPT := typDPT);
STLV59_563.STLV59_A_563_000.RB607_HVAC := M1_016_000_RB607_HVAC.xSwitch_OUT;
(* RB608_HVAC *)
(* RB609_HVAC *)
M1_017_000_RB608_HVAC(bPortKNX := 1, dwIndex_DPT := 17, typDPT := typDPT);
STLV59_563.STLV59_A_563_000.RB608_HVAC := M1_017_000_RB608_HVAC.xSwitch_OUT;
M1_018_000_RB609_HVAC(bPortKNX := 1, dwIndex_DPT := 18, typDPT := typDPT);
STLV59_563.STLV59_A_563_000.RB609_HVAC := M1_018_000_RB609_HVAC.xSwitch_OUT;
(* RT601_CT *)
(* RT602_CT *)
M1_019_000_RT601_CT(bPortKNX := 1, dwIndex_DPT := 19, typDPT := typDPT);
STLV59_563.STLV59_A_563_000.RT601_CT := M1_019_000_RT601_CT.rValue_OUT;
M1_020_000_RT602_CT(bPortKNX := 1, dwIndex_DPT := 20, typDPT := typDPT);
STLV59_563.STLV59_A_563_000.RT602_CT := M1_020_000_RT602_CT.rValue_OUT;
(* RT603_CT *)
(* RT604_CT *)
M1_021_000_RT603_CT(bPortKNX := 1, dwIndex_DPT := 21, typDPT := typDPT);
STLV59_563.STLV59_A_563_000.RT603_CT := M1_021_000_RT603_CT.rValue_OUT;
M1_022_000_RT604_CT(bPortKNX := 1, dwIndex_DPT := 22, typDPT := typDPT);
STLV59_563.STLV59_A_563_000.RT604_CT := M1_022_000_RT604_CT.rValue_OUT;
(* RT605_CT *)
(* RT606_CT *)
M1_023_000_RT605_CT(bPortKNX := 1, dwIndex_DPT := 23, typDPT := typDPT);
STLV59_563.STLV59_A_563_000.RT605_CT := M1_023_000_RT605_CT.rValue_OUT;
M1_024_000_RT606_CT(bPortKNX := 1, dwIndex_DPT := 24, typDPT := typDPT);
STLV59_563.STLV59_A_563_000.RT606_CT := M1_024_000_RT606_CT.rValue_OUT;
(* RT607_CT *)
(* RT608_CT *)
M1_025_000_RT607_CT(bPortKNX := 1, dwIndex_DPT := 25, typDPT := typDPT);
STLV59_563.STLV59_A_563_000.RT607_CT := M1_025_000_RT607_CT.rValue_OUT;
M1_026_000_RT608_CT(bPortKNX := 1, dwIndex_DPT := 26, typDPT := typDPT);
STLV59_563.STLV59_A_563_000.RT608_CT := M1_026_000_RT608_CT.rValue_OUT;
(* RT609_CT *)
(* RY601_CV *)
M1_027_000_RT609_CT(bPortKNX := 1, dwIndex_DPT := 27, typDPT := typDPT);
STLV59_563.STLV59_A_563_000.RT609_CT := M1_027_000_RT609_CT.rValue_OUT;
M1_028_000_RY601_CV(bPortKNX := 1, dwIndex_DPT := 28, typDPT := typDPT);
STLV59_563.STLV59_A_563_000.RY601_CV := M1_028_000_RY601_CV.rValue_OUT;
(* RY602_CV *)
(* RY603_CV *)
M1_029_000_RY602_CV(bPortKNX := 1, dwIndex_DPT := 29, typDPT := typDPT);
STLV59_563.STLV59_A_563_000.RY602_CV := M1_029_000_RY602_CV.rValue_OUT;
M1_030_000_RY603_CV(bPortKNX := 1, dwIndex_DPT := 30, typDPT := typDPT);
STLV59_563.STLV59_A_563_000.RY603_CV := M1_030_000_RY603_CV.rValue_OUT;
(* RY604_CV *)
(* RY605_CV *)
M1_031_000_RY604_CV(bPortKNX := 1, dwIndex_DPT := 31, typDPT := typDPT);
STLV59_563.STLV59_A_563_000.RY604_CV := M1_031_000_RY604_CV.rValue_OUT;
M1_032_000_RY605_CV(bPortKNX := 1, dwIndex_DPT := 32, typDPT := typDPT);
STLV59_563.STLV59_A_563_000.RY605_CV := M1_032_000_RY605_CV.rValue_OUT;
(* RY606_CV *)
(* RY607_CV *)
M1_033_000_RY606_CV(bPortKNX := 1, dwIndex_DPT := 33, typDPT := typDPT);
STLV59_563.STLV59_A_563_000.RY606_CV := M1_033_000_RY606_CV.rValue_OUT;
M1_034_000_RY607_CV(bPortKNX := 1, dwIndex_DPT := 34, typDPT := typDPT);
STLV59_563.STLV59_A_563_000.RY607_CV := M1_034_000_RY607_CV.rValue_OUT;
(* RY608_CV *)
(* RY609_CV *)
M1_035_000_RY608_CV(bPortKNX := 1, dwIndex_DPT := 35, typDPT := typDPT);
STLV59_563.STLV59_A_563_000.RY608_CV := M1_035_000_RY608_CV.rValue_OUT;
M1_036_000_RY609_CV(bPortKNX := 1, dwIndex_DPT := 36, typDPT := typDPT);
STLV59_563.STLV59_A_563_000.RY609_CV := M1_036_000_RY609_CV.rValue_OUT;
(* LH601_OP *)
(* LH602_OP *)
M1_037_000_LH601_OP(bPortKNX := 1, dwIndex_DPT := 37, rValue_IN := STLV59_563.STLV59_A_563_000.LH601_OP, xUpdate_KNX := i = 0, typDPT := typDPT);
M1_038_000_LH602_OP(bPortKNX := 1, dwIndex_DPT := 38, rValue_IN := STLV59_563.STLV59_A_563_000.LH602_OP, xUpdate_KNX := i = 1, typDPT := typDPT);
(* LH603_OP *)
(* LH604_OP *)
M1_039_000_LH603_OP(bPortKNX := 1, dwIndex_DPT := 39, rValue_IN := STLV59_563.STLV59_A_563_000.LH603_OP, xUpdate_KNX := i = 2, typDPT := typDPT);
M1_040_000_LH604_OP(bPortKNX := 1, dwIndex_DPT := 40, rValue_IN := STLV59_563.STLV59_A_563_000.LH604_OP, xUpdate_KNX := i = 3, typDPT := typDPT);
(* LH605_OP *)
(* LH606_OP *)
M1_041_000_LH605_OP(bPortKNX := 1, dwIndex_DPT := 41, rValue_IN := STLV59_563.STLV59_A_563_000.LH605_OP, xUpdate_KNX := i = 4, typDPT := typDPT);
M1_042_000_LH606_OP(bPortKNX := 1, dwIndex_DPT := 42, rValue_IN := STLV59_563.STLV59_A_563_000.LH606_OP, xUpdate_KNX := i = 5, typDPT := typDPT);
(* LH607_OP *)
(* LH608_OP *)
M1_043_000_LH607_OP(bPortKNX := 1, dwIndex_DPT := 43, rValue_IN := STLV59_563.STLV59_A_563_000.LH607_OP, xUpdate_KNX := i = 6, typDPT := typDPT);
M1_044_000_LH608_OP(bPortKNX := 1, dwIndex_DPT := 44, rValue_IN := STLV59_563.STLV59_A_563_000.LH608_OP, xUpdate_KNX := i = 7, typDPT := typDPT);
(* LH609_OP *)
(* LH601_CMD *)
M1_045_000_LH609_OP(bPortKNX := 1, dwIndex_DPT := 45, rValue_IN := STLV59_563.STLV59_A_563_000.LH609_OP, xUpdate_KNX := i = 8, typDPT := typDPT);
M1_046_000_LH601_CMD(bPortKNX := 1, dwIndex_DPT := 46, xSwitch_IN := STLV59_563.STLV59_A_563_000.LH601_CMD, xUpdate_KNX := i = 9, typDPT := typDPT);
(* LH602_CMD *)
(* LH603_CMD *)
M1_047_000_LH602_CMD(bPortKNX := 1, dwIndex_DPT := 47, xSwitch_IN := STLV59_563.STLV59_A_563_000.LH602_CMD, xUpdate_KNX := i = 10, typDPT := typDPT);
M1_048_000_LH603_CMD(bPortKNX := 1, dwIndex_DPT := 48, xSwitch_IN := STLV59_563.STLV59_A_563_000.LH603_CMD, xUpdate_KNX := i = 11, typDPT := typDPT);
(* LH604_CMD *)
(* LH605_CMD *)
M1_049_000_LH604_CMD(bPortKNX := 1, dwIndex_DPT := 49, xSwitch_IN := STLV59_563.STLV59_A_563_000.LH604_CMD, xUpdate_KNX := i = 12, typDPT := typDPT);
M1_050_000_LH605_CMD(bPortKNX := 1, dwIndex_DPT := 50, xSwitch_IN := STLV59_563.STLV59_A_563_000.LH605_CMD, xUpdate_KNX := i = 13, typDPT := typDPT);
(* LH606_CMD *)
(* LH607_CMD *)
M1_051_000_LH606_CMD(bPortKNX := 1, dwIndex_DPT := 51, xSwitch_IN := STLV59_563.STLV59_A_563_000.LH606_CMD, xUpdate_KNX := i = 14, typDPT := typDPT);
M1_052_000_LH607_CMD(bPortKNX := 1, dwIndex_DPT := 52, xSwitch_IN := STLV59_563.STLV59_A_563_000.LH607_CMD, xUpdate_KNX := i = 15, typDPT := typDPT);
(* LH608_CMD *)
(* LH609_CMD *)
M1_053_000_LH608_CMD(bPortKNX := 1, dwIndex_DPT := 53, xSwitch_IN := STLV59_563.STLV59_A_563_000.LH608_CMD, xUpdate_KNX := i = 16, typDPT := typDPT);
M1_054_000_LH609_CMD(bPortKNX := 1, dwIndex_DPT := 54, xSwitch_IN := STLV59_563.STLV59_A_563_000.LH609_CMD, xUpdate_KNX := i = 17, typDPT := typDPT);
(* LC601_OP *)
(* LC602_OP *)
M1_055_000_LC601_OP(bPortKNX := 1, dwIndex_DPT := 55, rValue_IN := STLV59_563.STLV59_A_563_000.LC601_OP, xUpdate_KNX := i = 18, typDPT := typDPT);
M1_056_000_LC602_OP(bPortKNX := 1, dwIndex_DPT := 56, rValue_IN := STLV59_563.STLV59_A_563_000.LC602_OP, xUpdate_KNX := i = 19, typDPT := typDPT);
(* LC603_OP *)
(* LC604_OP *)
M1_057_000_LC603_OP(bPortKNX := 1, dwIndex_DPT := 57, rValue_IN := STLV59_563.STLV59_A_563_000.LC603_OP, xUpdate_KNX := i = 20, typDPT := typDPT);
M1_058_000_LC604_OP(bPortKNX := 1, dwIndex_DPT := 58, rValue_IN := STLV59_563.STLV59_A_563_000.LC604_OP, xUpdate_KNX := i = 21, typDPT := typDPT);
(* LC605_OP *)
(* LC606_OP *)
M1_059_000_LC605_OP(bPortKNX := 1, dwIndex_DPT := 59, rValue_IN := STLV59_563.STLV59_A_563_000.LC605_OP, xUpdate_KNX := i = 22, typDPT := typDPT);
M1_060_000_LC606_OP(bPortKNX := 1, dwIndex_DPT := 60, rValue_IN := STLV59_563.STLV59_A_563_000.LC606_OP, xUpdate_KNX := i = 23, typDPT := typDPT);
(* LC607_OP *)
(* LC608_OP *)
M1_061_000_LC607_OP(bPortKNX := 1, dwIndex_DPT := 61, rValue_IN := STLV59_563.STLV59_A_563_000.LC607_OP, xUpdate_KNX := i = 24, typDPT := typDPT);
M1_062_000_LC608_OP(bPortKNX := 1, dwIndex_DPT := 62, rValue_IN := STLV59_563.STLV59_A_563_000.LC608_OP, xUpdate_KNX := i = 25, typDPT := typDPT);
(* LC609_OP *)
(* LC601_CMD *)
M1_063_000_LC609_OP(bPortKNX := 1, dwIndex_DPT := 63, rValue_IN := STLV59_563.STLV59_A_563_000.LC609_OP, xUpdate_KNX := i = 26, typDPT := typDPT);
M1_064_000_LC601_CMD(bPortKNX := 1, dwIndex_DPT := 64, xSwitch_IN := STLV59_563.STLV59_A_563_000.LC601_CMD, xUpdate_KNX := i = 27, typDPT := typDPT);
(* LC602_CMD *)
(* LC603_CMD *)
M1_065_000_LC602_CMD(bPortKNX := 1, dwIndex_DPT := 65, xSwitch_IN := STLV59_563.STLV59_A_563_000.LC602_CMD, xUpdate_KNX := i = 28, typDPT := typDPT);
M1_066_000_LC603_CMD(bPortKNX := 1, dwIndex_DPT := 66, xSwitch_IN := STLV59_563.STLV59_A_563_000.LC603_CMD, xUpdate_KNX := i = 29, typDPT := typDPT);
(* LC604_CMD *)
(* LC605_CMD *)
M1_067_000_LC604_CMD(bPortKNX := 1, dwIndex_DPT := 67, xSwitch_IN := STLV59_563.STLV59_A_563_000.LC604_CMD, xUpdate_KNX := i = 30, typDPT := typDPT);
M1_068_000_LC605_CMD(bPortKNX := 1, dwIndex_DPT := 68, xSwitch_IN := STLV59_563.STLV59_A_563_000.LC605_CMD, xUpdate_KNX := i = 31, typDPT := typDPT);
(* LC606_CMD *)
(* LC607_CMD *)
M1_069_000_LC606_CMD(bPortKNX := 1, dwIndex_DPT := 69, xSwitch_IN := STLV59_563.STLV59_A_563_000.LC606_CMD, xUpdate_KNX := i = 32, typDPT := typDPT);
M1_070_000_LC607_CMD(bPortKNX := 1, dwIndex_DPT := 70, xSwitch_IN := STLV59_563.STLV59_A_563_000.LC607_CMD, xUpdate_KNX := i = 33, typDPT := typDPT);
(* LC608_CMD *)
(* LC609_CMD *)
M1_071_000_LC608_CMD(bPortKNX := 1, dwIndex_DPT := 71, xSwitch_IN := STLV59_563.STLV59_A_563_000.LC608_CMD, xUpdate_KNX := i = 34, typDPT := typDPT);
M1_072_000_LC609_CMD(bPortKNX := 1, dwIndex_DPT := 72, xSwitch_IN := STLV59_563.STLV59_A_563_000.LC609_CMD, xUpdate_KNX := i = 35, typDPT := typDPT);
(* RT601_SP *)
(* RT602_SP *)
M1_073_000_RT601_SP(bPortKNX := 1, dwIndex_DPT := 73, rValue_IN := STLV59_563.STLV59_A_563_000.RT601_SP_D, xUpdate_KNX := NOT STLV59_563.STLV59_A_563_000.RB601_HVAC, typDPT := typDPT);
M1_074_000_RT602_SP(bPortKNX := 1, dwIndex_DPT := 74, rValue_IN := STLV59_563.STLV59_A_563_000.RT602_SP, xUpdate_KNX := NOT STLV59_563.STLV59_A_563_000.RB601_HVAC, typDPT := typDPT);
(* RT603_SP *)
(* RT604_SP *)
M1_075_000_RT603_SP(bPortKNX := 1, dwIndex_DPT := 75, rValue_IN := STLV59_563.STLV59_A_563_000.RT603_SP, xUpdate_KNX := NOT STLV59_563.STLV59_A_563_000.RB601_HVAC, typDPT := typDPT);
M1_076_000_RT604_SP(bPortKNX := 1, dwIndex_DPT := 76, rValue_IN := STLV59_563.STLV59_A_563_000.RT604_SP, xUpdate_KNX := NOT STLV59_563.STLV59_A_563_000.RB601_HVAC, typDPT := typDPT);
(* RT605_SP *)
(* RT606_SP *)
M1_077_000_RT605_SP(bPortKNX := 1, dwIndex_DPT := 77, rValue_IN := STLV59_563.STLV59_A_563_000.RT605_SP, xUpdate_KNX := NOT STLV59_563.STLV59_A_563_000.RB601_HVAC, typDPT := typDPT);
M1_078_000_RT606_SP(bPortKNX := 1, dwIndex_DPT := 78, rValue_IN := STLV59_563.STLV59_A_563_000.RT606_SP, xUpdate_KNX := NOT STLV59_563.STLV59_A_563_000.RB601_HVAC, typDPT := typDPT);
(* RT607_SP *)
(* RT608_SP *)
M1_079_000_RT607_SP(bPortKNX := 1, dwIndex_DPT := 79, rValue_IN := STLV59_563.STLV59_A_563_000.RT607_SP, xUpdate_KNX := NOT STLV59_563.STLV59_A_563_000.RB601_HVAC, typDPT := typDPT);
M1_080_000_RT608_SP(bPortKNX := 1, dwIndex_DPT := 80, rValue_IN := STLV59_563.STLV59_A_563_000.RT608_SP, xUpdate_KNX := NOT STLV59_563.STLV59_A_563_000.RB601_HVAC, typDPT := typDPT);
(* RT609_SP *)
(* RT601_SP Feedback *)
M1_081_000_RT609_SP(bPortKNX := 1, dwIndex_DPT := 81, rValue_IN := STLV59_563.STLV59_A_563_000.RT609_SP, xUpdate_KNX := NOT STLV59_563.STLV59_A_563_000.RB601_HVAC, typDPT := typDPT);
M1_082_000_RT601_SP_FB(bPortKNX := 1, dwIndex_DPT := 82, typDPT := typDPT);
STLV59_563.STLV59_A_563_000.RT601_SP_IN := M1_082_000_RT601_SP_FB.rValue_OUT;
(* RT602_SP Feedback *)
(* RT603_SP Feedback *)
M1_083_000_RT602_SP_FB(bPortKNX := 1, dwIndex_DPT := 83, typDPT := typDPT);
STLV59_563.STLV59_A_563_000.RT602_SP_IN := M1_083_000_RT602_SP_FB.rValue_OUT;
M1_084_000_RT603_SP_FB(bPortKNX := 1, dwIndex_DPT := 84, typDPT := typDPT);
STLV59_563.STLV59_A_563_000.RT603_SP_IN := M1_084_000_RT603_SP_FB.rValue_OUT;
(* RT604_SP Feedback *)
(* RT605_SP Feedback *)
M1_085_000_RT604_SP_FB(bPortKNX := 1, dwIndex_DPT := 85, typDPT := typDPT);
STLV59_563.STLV59_A_563_000.RT604_SP_IN := M1_085_000_RT604_SP_FB.rValue_OUT;
M1_086_000_RT605_SP_FB(bPortKNX := 1, dwIndex_DPT := 86, typDPT := typDPT);
STLV59_563.STLV59_A_563_000.RT605_SP_IN := M1_086_000_RT605_SP_FB.rValue_OUT;
(* RT606_SP Feedback *)
(* RT607_SP Feedback *)
M1_087_000_RT606_SP_FB(bPortKNX := 1, dwIndex_DPT := 87, typDPT := typDPT);
STLV59_563.STLV59_A_563_000.RT606_SP_IN := M1_087_000_RT606_SP_FB.rValue_OUT;
M1_088_000_RT607_SP_FB(bPortKNX := 1, dwIndex_DPT := 88, typDPT := typDPT);
STLV59_563.STLV59_A_563_000.RT607_SP_IN := M1_088_000_RT607_SP_FB.rValue_OUT;
(* RT608_SP Feedback *)
(* RT609_SP Feedback *)
M1_089_000_RT608_SP_FB(bPortKNX := 1, dwIndex_DPT := 89, typDPT := typDPT);
STLV59_563.STLV59_A_563_000.RT608_SP_IN := M1_089_000_RT608_SP_FB.rValue_OUT;
M1_090_000_RT609_SP_FB(bPortKNX := 1, dwIndex_DPT := 90, typDPT := typDPT);
STLV59_563.STLV59_A_563_000.RT609_SP_IN := M1_090_000_RT609_SP_FB.rValue_OUT;
(* LU601_V *)
(* LU602_V *)
M1_091_000_LU601_V(bPortKNX := 1, dwIndex_DPT := 91, typDPT := typDPT);
STLV59_563.STLV59_A_563_000.LU601_V := M1_091_000_LU601_V.xSwitch_OUT;
M1_092_000_LU602_V(bPortKNX := 1, dwIndex_DPT := 92, typDPT := typDPT);
STLV59_563.STLV59_A_563_000.LU602_V := M1_092_000_LU602_V.xSwitch_OUT;
(* LU603_V *)
(* LU604_V *)
M1_093_000_LU603_V(bPortKNX := 1, dwIndex_DPT := 93, typDPT := typDPT);
STLV59_563.STLV59_A_563_000.LU603_V := M1_093_000_LU603_V.xSwitch_OUT;
M1_094_000_LU604_V(bPortKNX := 1, dwIndex_DPT := 94, typDPT := typDPT);
STLV59_563.STLV59_A_563_000.LU604_V := M1_094_000_LU604_V.xSwitch_OUT;
(* LU605_V *)
(* LU606_V *)
M1_095_000_LU605_V(bPortKNX := 1, dwIndex_DPT := 95, typDPT := typDPT);
STLV59_563.STLV59_A_563_000.LU605_V := M1_095_000_LU605_V.xSwitch_OUT;
M1_096_000_LU606_V(bPortKNX := 1, dwIndex_DPT := 96, typDPT := typDPT);
STLV59_563.STLV59_A_563_000.LU606_V := M1_096_000_LU606_V.xSwitch_OUT;
(* LU607_V *)
(* LU608_V *)
M1_097_000_LU607_V(bPortKNX := 1, dwIndex_DPT := 97, typDPT := typDPT);
STLV59_563.STLV59_A_563_000.LU607_V := M1_097_000_LU607_V.xSwitch_OUT;
M1_098_000_LU608_V(bPortKNX := 1, dwIndex_DPT := 98, typDPT := typDPT);
STLV59_563.STLV59_A_563_000.LU608_V := M1_098_000_LU608_V.xSwitch_OUT;
(* LU609_V *)
(* LU601_AL *)
M1_099_000_LU609_V(bPortKNX := 1, dwIndex_DPT := 99, typDPT := typDPT);
STLV59_563.STLV59_A_563_000.LU609_V := M1_099_000_LU609_V.xSwitch_OUT;
M1_100_000_LU601_AL(bPortKNX := 1, dwIndex_DPT := 100, typDPT := typDPT);
STLV59_563.STLV59_A_563_000.LU601_AL := M1_100_000_LU601_AL.xSwitch_OUT;
(* LU602_AL *)
(* LU603_AL *)
M1_101_000_LU602_AL(bPortKNX := 1, dwIndex_DPT := 101, typDPT := typDPT);
STLV59_563.STLV59_A_563_000.LU602_AL := M1_101_000_LU602_AL.xSwitch_OUT;
M1_102_000_LU603_AL(bPortKNX := 1, dwIndex_DPT := 102, typDPT := typDPT);
STLV59_563.STLV59_A_563_000.LU603_AL := M1_102_000_LU603_AL.xSwitch_OUT;
(* LU604_AL *)
(* LU605_AL *)
M1_103_000_LU604_AL(bPortKNX := 1, dwIndex_DPT := 103, typDPT := typDPT);
STLV59_563.STLV59_A_563_000.LU604_AL := M1_103_000_LU604_AL.xSwitch_OUT;
M1_104_000_LU605_AL(bPortKNX := 1, dwIndex_DPT := 104, typDPT := typDPT);
STLV59_563.STLV59_A_563_000.LU605_AL := M1_104_000_LU605_AL.xSwitch_OUT;
(* LU606_AL *)
(* LU607_AL *)
M1_105_000_LU606_AL(bPortKNX := 1, dwIndex_DPT := 105, typDPT := typDPT);
STLV59_563.STLV59_A_563_000.LU606_AL := M1_105_000_LU606_AL.xSwitch_OUT;
M1_106_000_LU607_AL(bPortKNX := 1, dwIndex_DPT := 106, typDPT := typDPT);
STLV59_563.STLV59_A_563_000.LU607_AL := M1_106_000_LU607_AL.xSwitch_OUT;
(* LU608_AL *)
(* LU609_AL *)
M1_107_000_LU608_AL(bPortKNX := 1, dwIndex_DPT := 107, typDPT := typDPT);
STLV59_563.STLV59_A_563_000.LU608_AL := M1_107_000_LU608_AL.xSwitch_OUT;
M1_108_000_LU609_AL(bPortKNX := 1, dwIndex_DPT := 108, typDPT := typDPT);
STLV59_563.STLV59_A_563_000.LU609_AL := M1_108_000_LU609_AL.xSwitch_OUT;
(* LU601_CMD *)
(* LU602_CMD *)
M1_109_000_LU601_CMD(bPortKNX := 1, dwIndex_DPT := 109, xSwitch_IN := STLV59_563.STLV59_A_563_000.LU601_CMD, xUpdate_KNX := i = 36, typDPT := typDPT);
M1_110_000_LU602_CMD(bPortKNX := 1, dwIndex_DPT := 110, xSwitch_IN := STLV59_563.STLV59_A_563_000.LU602_CMD, xUpdate_KNX := i = 37, typDPT := typDPT);
(* LU603_CMD *)
(* LU604_CMD *)
M1_111_000_LU603_CMD(bPortKNX := 1, dwIndex_DPT := 111, xSwitch_IN := STLV59_563.STLV59_A_563_000.LU603_CMD, xUpdate_KNX := i = 38, typDPT := typDPT);
M1_112_000_LU604_CMD(bPortKNX := 1, dwIndex_DPT := 112, xSwitch_IN := STLV59_563.STLV59_A_563_000.LU604_CMD, xUpdate_KNX := i = 39, typDPT := typDPT);
(* LU605_CMD *)
(* LU606_CMD *)
M1_113_000_LU605_CMD(bPortKNX := 1, dwIndex_DPT := 113, xSwitch_IN := STLV59_563.STLV59_A_563_000.LU605_CMD, xUpdate_KNX := i = 40, typDPT := typDPT);
M1_114_000_LU606_CMD(bPortKNX := 1, dwIndex_DPT := 114, xSwitch_IN := STLV59_563.STLV59_A_563_000.LU606_CMD, xUpdate_KNX := i = 41, typDPT := typDPT);
(* LU607_CMD *)
(* LU608_CMD *)
M1_115_000_LU607_CMD(bPortKNX := 1, dwIndex_DPT := 115, xSwitch_IN := STLV59_563.STLV59_A_563_000.LU607_CMD, xUpdate_KNX := i = 42, typDPT := typDPT);
M1_116_000_LU608_CMD(bPortKNX := 1, dwIndex_DPT := 116, xSwitch_IN := STLV59_563.STLV59_A_563_000.LU608_CMD, xUpdate_KNX := i = 43, typDPT := typDPT);
(* LU609_CMD *)
M1_117_000_LU609_CMD(bPortKNX := 1, dwIndex_DPT := 117, xSwitch_IN := STLV59_563.STLV59_A_563_000.LU609_CMD, xUpdate_KNX := i = 44, typDPT := typDPT);
(* Rom 001 *)
(* RB601_V *)
(* RB602_V *)
M1_118_001_RB601_V(bPortKNX := 1, dwIndex_DPT := 118, typDPT := typDPT);
STLV59_563.STLV59_A_563_001.RB601_V := M1_118_001_RB601_V.xSwitch_OUT;
M1_119_001_RB602_V(bPortKNX := 1, dwIndex_DPT := 119, typDPT := typDPT);
STLV59_563.STLV59_A_563_001.RB602_V := M1_119_001_RB602_V.xSwitch_OUT;
(* RB601_HVAC *)
(* RB602_HVAC *)
M1_120_001_RB601_HVAC(bPortKNX := 1, dwIndex_DPT := 120, typDPT := typDPT);
STLV59_563.STLV59_A_563_001.RB601_HVAC := M1_120_001_RB601_HVAC.xSwitch_OUT;
M1_121_001_RB602_HVAC(bPortKNX := 1, dwIndex_DPT := 121, typDPT := typDPT);
STLV59_563.STLV59_A_563_001.RB602_HVAC := M1_121_001_RB602_HVAC.xSwitch_OUT;
(* RT601_CT *)
(* LH601_OP *)
M1_122_001_RT601_CT(bPortKNX := 1, dwIndex_DPT := 122, typDPT := typDPT);
STLV59_563.STLV59_A_563_001.RT601_CT := M1_122_001_RT601_CT.rValue_OUT;
M1_123_001_LH601_OP(bPortKNX := 1, dwIndex_DPT := 123, rValue_IN := STLV59_563.STLV59_A_563_001.LH601_OP, xUpdate_KNX := i = 45, typDPT := typDPT);
(* LH601_CMD *)
(* LC601_OP *)
M1_124_001_LH601_CMD(bPortKNX := 1, dwIndex_DPT := 124, xSwitch_IN := STLV59_563.STLV59_A_563_001.LH601_CMD, xUpdate_KNX := i = 46, typDPT := typDPT);
M1_125_001_LC601_OP(bPortKNX := 1, dwIndex_DPT := 125, rValue_IN := STLV59_563.STLV59_A_563_001.LC601_OP, xUpdate_KNX := i = 47, typDPT := typDPT);
(* LC601_CMD *)
(* LU601_V *)
M1_126_001_LC601_CMD(bPortKNX := 1, dwIndex_DPT := 126, xSwitch_IN := STLV59_563.STLV59_A_563_001.LC601_CMD, xUpdate_KNX := i = 48, typDPT := typDPT);
M1_127_001_LU601_V(bPortKNX := 1, dwIndex_DPT := 127, typDPT := typDPT);
STLV59_563.STLV59_A_563_001.LU601_V := M1_127_001_LU601_V.xSwitch_OUT;
(* LU601_AL *)
(* LU601_CMD *)
M1_128_001_LU601_AL(bPortKNX := 1, dwIndex_DPT := 128, typDPT := typDPT);
STLV59_563.STLV59_A_563_001.LU601_AL := M1_128_001_LU601_AL.xSwitch_OUT;
M1_129_001_LU601_CMD(bPortKNX := 1, dwIndex_DPT := 129, xSwitch_IN := STLV59_563.STLV59_A_563_001.LU601_CMD, xUpdate_KNX := i = 49, typDPT := typDPT);
(* Rom 002 *)
(* RB601_V *)
(* RB601_HVAC *)
M1_130_002_RB601_V(bPortKNX := 1, dwIndex_DPT := 130, typDPT := typDPT);
STLV59_563.STLV59_A_563_002.RB601_V := M1_130_002_RB601_V.xSwitch_OUT;
M1_131_002_RB601_HVAC(bPortKNX := 1, dwIndex_DPT := 131, typDPT := typDPT);
STLV59_563.STLV59_A_563_002.RB601_HVAC := M1_131_002_RB601_HVAC.xSwitch_OUT;
(* RT601_CT *)
(* RT602_CT *)
M1_132_002_RT601_CT(bPortKNX := 1, dwIndex_DPT := 132, typDPT := typDPT);
STLV59_563.STLV59_A_563_002.RT601_CT := M1_132_002_RT601_CT.rValue_OUT;
M1_133_002_RT602_CT(bPortKNX := 1, dwIndex_DPT := 133, typDPT := typDPT);
STLV59_563.STLV59_A_563_002.RT602_CT := M1_133_002_RT602_CT.rValue_OUT;
(* Rom 003 *)
(* RB601_V *)
(* RB601_HVAC *)
M1_134_003_RB601_V(bPortKNX := 1, dwIndex_DPT := 134, typDPT := typDPT);
STLV59_563.STLV59_A_563_003.RB601_V := M1_134_003_RB601_V.xSwitch_OUT;
M1_135_003_RB601_HVAC(bPortKNX := 1, dwIndex_DPT := 135, typDPT := typDPT);
STLV59_563.STLV59_A_563_003.RB601_HVAC := M1_135_003_RB601_HVAC.xSwitch_OUT;
(* Rom 004 *)
(* RB601_V *)
(* RB601_HVAC *)
M1_136_004_RB601_V(bPortKNX := 1, dwIndex_DPT := 136, typDPT := typDPT);
STLV59_563.STLV59_A_563_004.RB601_V := M1_136_004_RB601_V.xSwitch_OUT;
M1_137_004_RB601_HVAC(bPortKNX := 1, dwIndex_DPT := 137, typDPT := typDPT);
STLV59_563.STLV59_A_563_004.RB601_HVAC := M1_137_004_RB601_HVAC.xSwitch_OUT;
(* RT601_CT *)
(* RT602_CT *)
M1_138_004_RT601_CT(bPortKNX := 1, dwIndex_DPT := 138, typDPT := typDPT);
STLV59_563.STLV59_A_563_004.RT601_CT := M1_138_004_RT601_CT.rValue_OUT;
M1_139_004_RT602_CT(bPortKNX := 1, dwIndex_DPT := 139, typDPT := typDPT);
STLV59_563.STLV59_A_563_004.RT602_CT := M1_139_004_RT602_CT.rValue_OUT;
(* RY601_CV *)
M1_140_004_RY601_CV(bPortKNX := 1, dwIndex_DPT := 140, typDPT := typDPT);
STLV59_563.STLV59_A_563_004.RY601_CV := M1_140_004_RY601_CV.rValue_OUT;
(* Rom 005 *)
(* RB601_V *)
(* RB601_HVAC *)
M1_141_005_RB601_V(bPortKNX := 1, dwIndex_DPT := 141, typDPT := typDPT);
STLV59_563.STLV59_A_563_005.RB601_V := M1_141_005_RB601_V.xSwitch_OUT;
M1_142_005_RB601_HVAC(bPortKNX := 1, dwIndex_DPT := 142, typDPT := typDPT);
STLV59_563.STLV59_A_563_005.RB601_HVAC := M1_142_005_RB601_HVAC.xSwitch_OUT;
(* RT601_CT *)
(* RT602_CT *)
M1_143_005_RT601_CT(bPortKNX := 1, dwIndex_DPT := 143, typDPT := typDPT);
STLV59_563.STLV59_A_563_005.RT601_CT := M1_143_005_RT601_CT.rValue_OUT;
M1_144_005_RT602_CT(bPortKNX := 1, dwIndex_DPT := 144, typDPT := typDPT);
STLV59_563.STLV59_A_563_005.RT602_CT := M1_144_005_RT602_CT.rValue_OUT;
(* Rom 006 *)
(* RB601_V *)
(* RB601_HVAC *)
M1_145_006_RB601_V(bPortKNX := 1, dwIndex_DPT := 145, typDPT := typDPT);
STLV59_563.STLV59_A_563_006.RB601_V := M1_145_006_RB601_V.xSwitch_OUT;
M1_146_006_RB601_HVAC(bPortKNX := 1, dwIndex_DPT := 146, typDPT := typDPT);
STLV59_563.STLV59_A_563_006.RB601_HVAC := M1_146_006_RB601_HVAC.xSwitch_OUT;
(* RT601_CT *)
M1_147_006_RT601_CT(bPortKNX := 1, dwIndex_DPT := 147, typDPT := typDPT);
STLV59_563.STLV59_A_563_006.RT601_CT := M1_147_006_RT601_CT.rValue_OUT;
(* Rom 007 *)
(* RB601_V *)
(* RB601_HVAC *)
M1_148_007_RB601_V(bPortKNX := 1, dwIndex_DPT := 148, typDPT := typDPT);
STLV59_563.STLV59_A_563_007.RB601_V := M1_148_007_RB601_V.xSwitch_OUT;
M1_149_007_RB601_HVAC(bPortKNX := 1, dwIndex_DPT := 149, typDPT := typDPT);
STLV59_563.STLV59_A_563_007.RB601_HVAC := M1_149_007_RB601_HVAC.xSwitch_OUT;
(* RT601_CT *)
(* RT602_CT *)
M1_150_007_RT601_CT(bPortKNX := 1, dwIndex_DPT := 150, typDPT := typDPT);
STLV59_563.STLV59_A_563_007.RT601_CT := M1_150_007_RT601_CT.rValue_OUT;
M1_151_007_RT602_CT(bPortKNX := 1, dwIndex_DPT := 151, typDPT := typDPT);
STLV59_563.STLV59_A_563_007.RT602_CT := M1_151_007_RT602_CT.rValue_OUT;
(* Rom 008 *)
(* RB601_V *)
(* RB601_HVAC *)
M1_152_008_RB601_V(bPortKNX := 1, dwIndex_DPT := 152, typDPT := typDPT);
STLV59_563.STLV59_A_563_008.RB601_V := M1_152_008_RB601_V.xSwitch_OUT;
M1_153_008_RB601_HVAC(bPortKNX := 1, dwIndex_DPT := 153, typDPT := typDPT);
STLV59_563.STLV59_A_563_008.RB601_HVAC := M1_153_008_RB601_HVAC.xSwitch_OUT;
(* RT601_CT *)
(* RT602_CT *)
M1_154_008_RT601_CT(bPortKNX := 1, dwIndex_DPT := 154, typDPT := typDPT);
STLV59_563.STLV59_A_563_008.RT601_CT := M1_154_008_RT601_CT.rValue_OUT;
M1_155_008_RT602_CT(bPortKNX := 1, dwIndex_DPT := 155, typDPT := typDPT);
STLV59_563.STLV59_A_563_008.RT602_CT := M1_155_008_RT602_CT.rValue_OUT;
(* Rom 009 *)
(* RB601_V *)
(* RB601_HVAC *)
M1_156_009_RB601_V(bPortKNX := 1, dwIndex_DPT := 156, typDPT := typDPT);
STLV59_563.STLV59_A_563_009.RB601_V := M1_156_009_RB601_V.xSwitch_OUT;
M1_157_009_RB601_HVAC(bPortKNX := 1, dwIndex_DPT := 157, typDPT := typDPT);
STLV59_563.STLV59_A_563_009.RB601_HVAC := M1_157_009_RB601_HVAC.xSwitch_OUT;
(* RT601_CT *)
(* RT602_CT *)
M1_158_009_RT601_CT(bPortKNX := 1, dwIndex_DPT := 158, typDPT := typDPT);
STLV59_563.STLV59_A_563_009.RT601_CT := M1_158_009_RT601_CT.rValue_OUT;
M1_159_009_RT602_CT(bPortKNX := 1, dwIndex_DPT := 159, typDPT := typDPT);
STLV59_563.STLV59_A_563_009.RT602_CT := M1_159_009_RT602_CT.rValue_OUT;
(* Rom 010 *)
(* RB601_V *)
(* RB601_HVAC *)
M1_160_010_RB601_V(bPortKNX := 1, dwIndex_DPT := 160, typDPT := typDPT);
STLV59_563.STLV59_A_563_010.RB601_V := M1_160_010_RB601_V.xSwitch_OUT;
M1_161_010_RB601_HVAC(bPortKNX := 1, dwIndex_DPT := 161, typDPT := typDPT);
STLV59_563.STLV59_A_563_010.RB601_HVAC := M1_161_010_RB601_HVAC.xSwitch_OUT;
(* RT601_CT *)
(* RT602_CT *)
M1_162_010_RT601_CT(bPortKNX := 1, dwIndex_DPT := 162, typDPT := typDPT);
STLV59_563.STLV59_A_563_010.RT601_CT := M1_162_010_RT601_CT.rValue_OUT;
M1_163_010_RT602_CT(bPortKNX := 1, dwIndex_DPT := 163, typDPT := typDPT);
STLV59_563.STLV59_A_563_010.RT602_CT := M1_163_010_RT602_CT.rValue_OUT;
(* Rom 011 *)
(* RB601_V *)
(* RB601_HVAC *)
M1_164_011_RB601_V(bPortKNX := 1, dwIndex_DPT := 164, typDPT := typDPT);
STLV59_563.STLV59_A_563_011.RB601_V := M1_164_011_RB601_V.xSwitch_OUT;
M1_165_011_RB601_HVAC(bPortKNX := 1, dwIndex_DPT := 165, typDPT := typDPT);
STLV59_563.STLV59_A_563_011.RB601_HVAC := M1_165_011_RB601_HVAC.xSwitch_OUT;
(* RT601_CT *)
(* RT602_CT *)
M1_166_011_RT601_CT(bPortKNX := 1, dwIndex_DPT := 166, typDPT := typDPT);
STLV59_563.STLV59_A_563_011.RT601_CT := M1_166_011_RT601_CT.rValue_OUT;
M1_167_011_RT602_CT(bPortKNX := 1, dwIndex_DPT := 167, typDPT := typDPT);
STLV59_563.STLV59_A_563_011.RT602_CT := M1_167_011_RT602_CT.rValue_OUT;
(* Rom 012 *)
(* RB601_V *)
(* RB601_HVAC *)
M1_168_012_RB601_V(bPortKNX := 1, dwIndex_DPT := 168, typDPT := typDPT);
STLV59_563.STLV59_A_563_012.RB601_V := M1_168_012_RB601_V.xSwitch_OUT;
M1_169_012_RB601_HVAC(bPortKNX := 1, dwIndex_DPT := 169, typDPT := typDPT);
STLV59_563.STLV59_A_563_012.RB601_HVAC := M1_169_012_RB601_HVAC.xSwitch_OUT;
(* RT601_CT *)
(* RT602_CT *)
M1_170_012_RT601_CT(bPortKNX := 1, dwIndex_DPT := 170, typDPT := typDPT);
STLV59_563.STLV59_A_563_012.RT601_CT := M1_170_012_RT601_CT.rValue_OUT;
M1_171_012_RT602_CT(bPortKNX := 1, dwIndex_DPT := 171, typDPT := typDPT);
STLV59_563.STLV59_A_563_012.RT602_CT := M1_171_012_RT602_CT.rValue_OUT;
(* Rom 013 *)
(* RB601_V *)
(* RB601_HVAC *)
M1_172_013_RB601_V(bPortKNX := 1, dwIndex_DPT := 172, typDPT := typDPT);
STLV59_563.STLV59_A_563_013.RB601_V := M1_172_013_RB601_V.xSwitch_OUT;
M1_173_013_RB601_HVAC(bPortKNX := 1, dwIndex_DPT := 173, typDPT := typDPT);
STLV59_563.STLV59_A_563_013.RB601_HVAC := M1_173_013_RB601_HVAC.xSwitch_OUT;
(* RT601_CT *)
(* RT602_CT *)
M1_174_013_RT601_CT(bPortKNX := 1, dwIndex_DPT := 174, typDPT := typDPT);
STLV59_563.STLV59_A_563_013.RT601_CT := M1_174_013_RT601_CT.rValue_OUT;
M1_175_013_RT602_CT(bPortKNX := 1, dwIndex_DPT := 175, typDPT := typDPT);
STLV59_563.STLV59_A_563_013.RT602_CT := M1_175_013_RT602_CT.rValue_OUT;
(* Rom 014 *)
(* RB601_V *)
(* RB602_V *)
M1_176_014_RB601_V(bPortKNX := 1, dwIndex_DPT := 176, typDPT := typDPT);
STLV59_563.STLV59_A_563_014.RB601_V := M1_176_014_RB601_V.xSwitch_OUT;
M1_177_014_RB602_V(bPortKNX := 1, dwIndex_DPT := 177, typDPT := typDPT);
STLV59_563.STLV59_A_563_014.RB602_V := M1_177_014_RB602_V.xSwitch_OUT;
(* RB601_HVAC *)
(* RB602_HVAC *)
M1_178_014_RB601_HVAC(bPortKNX := 1, dwIndex_DPT := 178, typDPT := typDPT);
STLV59_563.STLV59_A_563_014.RB601_HVAC := M1_178_014_RB601_HVAC.xSwitch_OUT;
M1_179_014_RB602_HVAC(bPortKNX := 1, dwIndex_DPT := 179, typDPT := typDPT);
STLV59_563.STLV59_A_563_014.RB602_HVAC := M1_179_014_RB602_HVAC.xSwitch_OUT;
(* Rom 015 *)
(* RB601_V *)
(* RB601_HVAC *)
M1_180_015_RB601_V(bPortKNX := 1, dwIndex_DPT := 180, typDPT := typDPT);
STLV59_563.STLV59_A_563_015.RB601_V := M1_180_015_RB601_V.xSwitch_OUT;
M1_181_015_RB601_HVAC(bPortKNX := 1, dwIndex_DPT := 181, typDPT := typDPT);
STLV59_563.STLV59_A_563_015.RB601_HVAC := M1_181_015_RB601_HVAC.xSwitch_OUT;
(* Rom 016 *)
(* RB601_V *)
(* RB601_HVAC *)
M1_182_016_RB601_V(bPortKNX := 1, dwIndex_DPT := 182, typDPT := typDPT);
STLV59_563.STLV59_A_563_016.RB601_V := M1_182_016_RB601_V.xSwitch_OUT;
M1_183_016_RB601_HVAC(bPortKNX := 1, dwIndex_DPT := 183, typDPT := typDPT);
STLV59_563.STLV59_A_563_016.RB601_HVAC := M1_183_016_RB601_HVAC.xSwitch_OUT;
(* Rom 017 *)
(* RB601_V *)
(* RB601_HVAC *)
M1_184_017_RB601_V(bPortKNX := 1, dwIndex_DPT := 184, typDPT := typDPT);
STLV59_563.STLV59_A_563_017.RB601_V := M1_184_017_RB601_V.xSwitch_OUT;
M1_185_017_RB601_HVAC(bPortKNX := 1, dwIndex_DPT := 185, typDPT := typDPT);
STLV59_563.STLV59_A_563_017.RB601_HVAC := M1_185_017_RB601_HVAC.xSwitch_OUT;
(* RT601_CT *)
(* RT602_CT *)
M1_186_017_RT601_CT(bPortKNX := 1, dwIndex_DPT := 186, typDPT := typDPT);
STLV59_563.STLV59_A_563_017.RT601_CT := M1_186_017_RT601_CT.rValue_OUT;
M1_187_017_RT602_CT(bPortKNX := 1, dwIndex_DPT := 187, typDPT := typDPT);
STLV59_563.STLV59_A_563_017.RT602_CT := M1_187_017_RT602_CT.rValue_OUT;
(* Rom 101 *)
(* RB601_V *)
(* RB601_HVAC *)
M1_188_101_RB601_V(bPortKNX := 1, dwIndex_DPT := 188, typDPT := typDPT);
STLV59_563.STLV59_A_563_101.RB601_V := M1_188_101_RB601_V.xSwitch_OUT;
M1_189_101_RB601_HVAC(bPortKNX := 1, dwIndex_DPT := 189, typDPT := typDPT);
STLV59_563.STLV59_A_563_101.RB601_HVAC := M1_189_101_RB601_HVAC.xSwitch_OUT;
(* RT601_CT *)
(* RT602_CT *)
M1_190_101_RT601_CT(bPortKNX := 1, dwIndex_DPT := 190, typDPT := typDPT);
STLV59_563.STLV59_A_563_101.RT601_CT := M1_190_101_RT601_CT.rValue_OUT;
M1_191_101_RT602_CT(bPortKNX := 1, dwIndex_DPT := 191, typDPT := typDPT);
STLV59_563.STLV59_A_563_101.RT602_CT := M1_191_101_RT602_CT.rValue_OUT;
(* Rom 102 *)
(* RB601_V *)
(* RB601_HVAC *)
M1_192_102_RB601_V(bPortKNX := 1, dwIndex_DPT := 192, typDPT := typDPT);
STLV59_563.STLV59_A_563_102.RB601_V := M1_192_102_RB601_V.xSwitch_OUT;
M1_193_102_RB601_HVAC(bPortKNX := 1, dwIndex_DPT := 193, typDPT := typDPT);
STLV59_563.STLV59_A_563_102.RB601_HVAC := M1_193_102_RB601_HVAC.xSwitch_OUT;
(* RT601_CT *)
(* RT602_CT *)
M1_194_102_RT601_CT(bPortKNX := 1, dwIndex_DPT := 194, typDPT := typDPT);
STLV59_563.STLV59_A_563_102.RT601_CT := M1_194_102_RT601_CT.rValue_OUT;
M1_195_102_RT602_CT(bPortKNX := 1, dwIndex_DPT := 195, typDPT := typDPT);
STLV59_563.STLV59_A_563_102.RT602_CT := M1_195_102_RT602_CT.rValue_OUT;
(* Rom 103 *)
(* RB601_V *)
(* RB602_V *)
M1_196_103_RB601_V(bPortKNX := 1, dwIndex_DPT := 196, typDPT := typDPT);
STLV59_563.STLV59_A_563_103.RB601_V := M1_196_103_RB601_V.xSwitch_OUT;
M1_197_103_RB602_V(bPortKNX := 1, dwIndex_DPT := 197, typDPT := typDPT);
STLV59_563.STLV59_A_563_103.RB602_V := M1_197_103_RB602_V.xSwitch_OUT;
(* RB603_V *)
(* RB604_V *)
M1_198_103_RB603_V(bPortKNX := 1, dwIndex_DPT := 198, typDPT := typDPT);
STLV59_563.STLV59_A_563_103.RB603_V := M1_198_103_RB603_V.xSwitch_OUT;
M1_199_103_RB604_V(bPortKNX := 1, dwIndex_DPT := 199, typDPT := typDPT);
STLV59_563.STLV59_A_563_103.RB604_V := M1_199_103_RB604_V.xSwitch_OUT;
(* RB601_HVAC *)
(* RB602_HVAC *)
M1_200_103_RB601_HVAC(bPortKNX := 1, dwIndex_DPT := 200, typDPT := typDPT);
STLV59_563.STLV59_A_563_103.RB601_HVAC := M1_200_103_RB601_HVAC.xSwitch_OUT;
M1_201_103_RB602_HVAC(bPortKNX := 1, dwIndex_DPT := 201, typDPT := typDPT);
STLV59_563.STLV59_A_563_103.RB602_HVAC := M1_201_103_RB602_HVAC.xSwitch_OUT;
(* RB603_HVAC *)
(* RB604_HVAC *)
M1_202_103_RB603_HVAC(bPortKNX := 1, dwIndex_DPT := 202, typDPT := typDPT);
STLV59_563.STLV59_A_563_103.RB603_HVAC := M1_202_103_RB603_HVAC.xSwitch_OUT;
M1_203_103_RB604_HVAC(bPortKNX := 1, dwIndex_DPT := 203, typDPT := typDPT);
STLV59_563.STLV59_A_563_103.RB604_HVAC := M1_203_103_RB604_HVAC.xSwitch_OUT;
(* RT601_CT *)
(* RT602_CT *)
M1_204_103_RT601_CT(bPortKNX := 1, dwIndex_DPT := 204, typDPT := typDPT);
STLV59_563.STLV59_A_563_103.RT601_CT := M1_204_103_RT601_CT.rValue_OUT;
M1_205_103_RT602_CT(bPortKNX := 1, dwIndex_DPT := 205, typDPT := typDPT);
STLV59_563.STLV59_A_563_103.RT602_CT := M1_205_103_RT602_CT.rValue_OUT;
(* RY601_CV *)
M1_206_103_RY601_CV(bPortKNX := 1, dwIndex_DPT := 206, typDPT := typDPT);
STLV59_563.STLV59_A_563_103.RY601_CV := M1_206_103_RY601_CV.rValue_OUT;
(* Rom 109 *)
(* RB601_V *)
(* RB601_HVAC *)
M1_207_109_RB601_V(bPortKNX := 1, dwIndex_DPT := 207, typDPT := typDPT);
STLV59_563.STLV59_A_563_109.RB601_V := M1_207_109_RB601_V.xSwitch_OUT;
M1_208_109_RB601_HVAC(bPortKNX := 1, dwIndex_DPT := 208, typDPT := typDPT);
STLV59_563.STLV59_A_563_109.RB601_HVAC := M1_208_109_RB601_HVAC.xSwitch_OUT;
(* RT601_CT *)
(* RT602_CT *)
M1_209_109_RT601_CT(bPortKNX := 1, dwIndex_DPT := 209, typDPT := typDPT);
STLV59_563.STLV59_A_563_109.RT601_CT := M1_209_109_RT601_CT.rValue_OUT;
M1_210_109_RT602_CT(bPortKNX := 1, dwIndex_DPT := 210, typDPT := typDPT);
STLV59_563.STLV59_A_563_109.RT602_CT := M1_210_109_RT602_CT.rValue_OUT;
(* Rom 201 *)
(* RT601_CT *)
(* RT602_CT *)
M1_211_201_RT601_CT(bPortKNX := 1, dwIndex_DPT := 211, typDPT := typDPT);
STLV59_563.STLV59_A_563_201.RT601_CT := M1_211_201_RT601_CT.rValue_OUT;
M1_212_201_RT602_CT(bPortKNX := 1, dwIndex_DPT := 212, typDPT := typDPT);
STLV59_563.STLV59_A_563_201.RT602_CT := M1_212_201_RT602_CT.rValue_OUT;
(* RT603_CT *)
M1_213_201_RT603_CT(bPortKNX := 1, dwIndex_DPT := 213, typDPT := typDPT);
STLV59_563.STLV59_A_563_201.RT603_CT := M1_213_201_RT603_CT.rValue_OUT;
(* Rom 212 *)
(* RB601_V *)
(* RB601_HVAC *)
M1_214_212_RB601_V(bPortKNX := 1, dwIndex_DPT := 214, typDPT := typDPT);
STLV59_563.STLV59_A_563_212.RB601_V := M1_214_212_RB601_V.xSwitch_OUT;
M1_215_212_RB601_HVAC(bPortKNX := 1, dwIndex_DPT := 215, typDPT := typDPT);
STLV59_563.STLV59_A_563_212.RB601_HVAC := M1_215_212_RB601_HVAC.xSwitch_OUT;
(* RT601_CT *)
(* RT602_CT *)
M1_216_212_RT601_CT(bPortKNX := 1, dwIndex_DPT := 216, typDPT := typDPT);
STLV59_563.STLV59_A_563_212.RT601_CT := M1_216_212_RT601_CT.rValue_OUT;
M1_217_212_RT602_CT(bPortKNX := 1, dwIndex_DPT := 217, typDPT := typDPT);
STLV59_563.STLV59_A_563_212.RT602_CT := M1_217_212_RT602_CT.rValue_OUT;
(* RY601_CV *)
M1_218_212_RY601_CV(bPortKNX := 1, dwIndex_DPT := 218, typDPT := typDPT);
STLV59_563.STLV59_A_563_212.RY601_CV := M1_218_212_RY601_CV.rValue_OUT;
(* Rom 213 *)
(* RB601_V *)
(* RB601_HVAC *)
M1_219_213_RB601_V(bPortKNX := 1, dwIndex_DPT := 219, typDPT := typDPT);
STLV59_563.STLV59_A_563_213.RB601_V := M1_219_213_RB601_V.xSwitch_OUT;
M1_220_213_RB601_HVAC(bPortKNX := 1, dwIndex_DPT := 220, typDPT := typDPT);
STLV59_563.STLV59_A_563_213.RB601_HVAC := M1_220_213_RB601_HVAC.xSwitch_OUT;
(* RT601_CT *)
(* RT602_CT *)
M1_221_213_RT601_CT(bPortKNX := 1, dwIndex_DPT := 221, typDPT := typDPT);
STLV59_563.STLV59_A_563_213.RT601_CT := M1_221_213_RT601_CT.rValue_OUT;
M1_222_213_RT602_CT(bPortKNX := 1, dwIndex_DPT := 222, typDPT := typDPT);
STLV59_563.STLV59_A_563_213.RT602_CT := M1_222_213_RT602_CT.rValue_OUT;
(* Rom T2_1 *)
(* RB601_V *)
(* RB601_HVAC *)
M1_223_T2_1_RB601_V(bPortKNX := 1, dwIndex_DPT := 223, typDPT := typDPT);
STLV59_563.STLV59_A_563_T2_1.RB601_V := M1_223_T2_1_RB601_V.xSwitch_OUT;
M1_224_T2_1_RB601_HVAC(bPortKNX := 1, dwIndex_DPT := 224, typDPT := typDPT);
STLV59_563.STLV59_A_563_T2_1.RB601_HVAC := M1_224_T2_1_RB601_HVAC.xSwitch_OUT;
(* RT601_CT *)
(* RT602_CT *)
M1_225_T2_1_RT601_CT(bPortKNX := 1, dwIndex_DPT := 225, typDPT := typDPT);
STLV59_563.STLV59_A_563_T2_1.RT601_CT := M1_225_T2_1_RT601_CT.rValue_OUT;
M1_226_T2_1_RT602_CT(bPortKNX := 1, dwIndex_DPT := 226, typDPT := typDPT);
STLV59_563.STLV59_A_563_T2_1.RT602_CT := M1_226_T2_1_RT602_CT.rValue_OUT;
(* Rom T2_2 *)
(* RB601_V *)
(* RB601_HVAC *)
M1_227_T2_2_RB601_V(bPortKNX := 1, dwIndex_DPT := 227, typDPT := typDPT);
STLV59_563.STLV59_A_563_T2_2.RB601_V := M1_227_T2_2_RB601_V.xSwitch_OUT;
M1_228_T2_2_RB601_HVAC(bPortKNX := 1, dwIndex_DPT := 228, typDPT := typDPT);
STLV59_563.STLV59_A_563_T2_2.RB601_HVAC := M1_228_T2_2_RB601_HVAC.xSwitch_OUT;
(* RT601_CT *)
(* RT602_CT *)
M1_229_T2_2_RT601_CT(bPortKNX := 1, dwIndex_DPT := 229, typDPT := typDPT);
STLV59_563.STLV59_A_563_T2_2.RT601_CT := M1_229_T2_2_RT601_CT.rValue_OUT;
M1_230_T2_2_RT602_CT(bPortKNX := 1, dwIndex_DPT := 230, typDPT := typDPT);
STLV59_563.STLV59_A_563_T2_2.RT602_CT := M1_230_T2_2_RT602_CT.rValue_OUT;
END_PROGRAM

PROGRAM PRG_563_Romstyring
  VAR
    Rom_000 : fbRomtype_99999999999999;  (* 000 *)
    Rom_001 : fbRomtype_2210111100111;  (* 001 *)
    Rom_002 : fbRomtype_1120011;  (* 002 *)
    Rom_004 : fbRomtype_1121;  (* 004 *)
    Rom_005 : fbRomtype_112001;  (* 005 *)
    Rom_007 : fbRomtype_112001;  (* 007 *)
    Rom_008 : fbRomtype_112001;  (* 008 *)
    Rom_009 : fbRomtype_112001;  (* 009 *)
    Rom_010 : fbRomtype_112001;  (* 010 *)
    Rom_011 : fbRomtype_112001;  (* 011 *)
    Rom_012 : fbRomtype_112001;  (* 012 *)
    Rom_013 : fbRomtype_112001;  (* 013 *)
    Rom_017 : fbRomtype_112001;  (* 017 *)
    Rom_101 : fbRomtype_112001;  (* 101 *)
    Rom_102 : fbRomtype_112001;  (* 102 *)
    Rom_103 : fbRomtype_4421011;  (* 103 *)
    Rom_109 : fbRomtype_112001;  (* 109 *)
    Rom_212 : fbRomtype_1121011;  (* 212 *)
    Rom_T2_1 : fbRomtype_112001;  (* T2_1 *)
    Rom_T2_2 : fbRomtype_112001;  (* T2_2 *)
  END_VAR

(* CFC diagram, written out as Structured Text *)
(* Rom 000 *)
Rom_000(RB601_HVAC := STLV59_563.STLV59_A_563_000.RB601_HVAC, RB602_HVAC := STLV59_563.STLV59_A_563_000.RB602_HVAC, RB603_HVAC := STLV59_563.STLV59_A_563_000.RB603_HVAC, RB604_HVAC := STLV59_563.STLV59_A_563_000.RB604_HVAC, RB605_HVAC := STLV59_563.STLV59_A_563_000.RB605_HVAC, RB606_HVAC := STLV59_563.STLV59_A_563_000.RB606_HVAC, RB607_HVAC := STLV59_563.STLV59_A_563_000.RB607_HVAC, RB608_HVAC := STLV59_563.STLV59_A_563_000.RB608_HVAC, RB609_HVAC := STLV59_563.STLV59_A_563_000.RB609_HVAC, RT601_CT := STLV59_563.STLV59_A_563_000.RT601_CT, RT602_CT := STLV59_563.STLV59_A_563_000.RT602_CT, RT602_SP := STLV59_563.STLV59_A_563_000.RT602_SP, RT603_CT := STLV59_563.STLV59_A_563_000.RT603_CT, RT603_SP := STLV59_563.STLV59_A_563_000.RT603_SP, RT604_CT := STLV59_563.STLV59_A_563_000.RT604_CT, RT604_SP := STLV59_563.STLV59_A_563_000.RT604_SP, RT605_CT := STLV59_563.STLV59_A_563_000.RT605_CT, RT605_SP := STLV59_563.STLV59_A_563_000.RT605_SP, RT606_CT := STLV59_563.STLV59_A_563_000.RT606_CT, RT606_SP := STLV59_563.STLV59_A_563_000.RT606_SP, RT607_CT := STLV59_563.STLV59_A_563_000.RT607_CT, RT607_SP := STLV59_563.STLV59_A_563_000.RT607_SP, RT608_CT := STLV59_563.STLV59_A_563_000.RT608_CT, RT608_SP := STLV59_563.STLV59_A_563_000.RT608_SP, RT609_CT := STLV59_563.STLV59_A_563_000.RT609_CT, RT609_SP := STLV59_563.STLV59_A_563_000.RT609_SP, RT601_SP_D := STLV59_563.STLV59_A_563_000.RT601_SP_D, RT601_SP_S := STLV59_563.STLV59_A_563_000.RT601_SP_S, RT601_SP_N := STLV59_563.STLV59_A_563_000.RT601_SP_N, RT601_SP_F := STLV59_563.STLV59_A_563_000.RT601_SP_F, OPM := STLV59_563.STLV59_A_563_000.OPM, RY601_CV := STLV59_563.STLV59_A_563_000.RY601_CV, RY602_CV := STLV59_563.STLV59_A_563_000.RY602_CV, RY603_CV := STLV59_563.STLV59_A_563_000.RY603_CV, RY604_CV := STLV59_563.STLV59_A_563_000.RY604_CV, RY605_CV := STLV59_563.STLV59_A_563_000.RY605_CV, RY606_CV := STLV59_563.STLV59_A_563_000.RY606_CV, RY607_CV := STLV59_563.STLV59_A_563_000.RY607_CV, RY608_CV := STLV59_563.STLV59_A_563_000.RY608_CV, RY609_CV := STLV59_563.STLV59_A_563_000.RY609_CV, RY601_SP := STLV59_563.STLV59_A_563_000.RY601_SP, LH601_MAN := STLV59_563.STLV59_A_563_000.LH601_MAN, LC601_MAN := STLV59_563.STLV59_A_563_000.LC601_MAN, RT601_SP_IN := STLV59_563.STLV59_A_563_000.RT601_SP_IN, RT602_SP_IN := STLV59_563.STLV59_A_563_000.RT602_SP_IN, RT603_SP_IN := STLV59_563.STLV59_A_563_000.RT603_SP_IN, RT604_SP_IN := STLV59_563.STLV59_A_563_000.RT604_SP_IN, RT605_SP_IN := STLV59_563.STLV59_A_563_000.RT605_SP_IN, RT606_SP_IN := STLV59_563.STLV59_A_563_000.RT606_SP_IN, RT607_SP_IN := STLV59_563.STLV59_A_563_000.RT607_SP_IN, RT608_SP_IN := STLV59_563.STLV59_A_563_000.RT608_SP_IN, RT609_SP_IN := STLV59_563.STLV59_A_563_000.RT609_SP_IN, LU601_V := STLV59_563.STLV59_A_563_000.LU601_V, LU602_V := STLV59_563.STLV59_A_563_000.LU602_V, LU603_V := STLV59_563.STLV59_A_563_000.LU603_V, LU604_V := STLV59_563.STLV59_A_563_000.LU604_V, LU605_V := STLV59_563.STLV59_A_563_000.LU605_V, LU606_V := STLV59_563.STLV59_A_563_000.LU606_V, LU607_V := STLV59_563.STLV59_A_563_000.LU607_V, LU608_V := STLV59_563.STLV59_A_563_000.LU608_V, LU609_V := STLV59_563.STLV59_A_563_000.LU609_V);
STLV59_563.STLV59_A_563_000.OPM_CV := Rom_000.OPM_CV;
STLV59_563.STLV59_A_563_000.RT601_CS := Rom_000.RT601_CS;
STLV59_563.STLV59_A_563_000.RY601_OP := Rom_000.RY601_OP;
STLV59_563.STLV59_A_563_000.LH601_OP := Rom_000.LH601_OP;
STLV59_563.STLV59_A_563_000.LH602_OP := Rom_000.LH602_OP;
STLV59_563.STLV59_A_563_000.LH603_OP := Rom_000.LH603_OP;
STLV59_563.STLV59_A_563_000.LH604_OP := Rom_000.LH604_OP;
STLV59_563.STLV59_A_563_000.LH605_OP := Rom_000.LH605_OP;
STLV59_563.STLV59_A_563_000.LH606_OP := Rom_000.LH606_OP;
STLV59_563.STLV59_A_563_000.LH607_OP := Rom_000.LH607_OP;
STLV59_563.STLV59_A_563_000.LH608_OP := Rom_000.LH608_OP;
STLV59_563.STLV59_A_563_000.LH609_OP := Rom_000.LH609_OP;
STLV59_563.STLV59_A_563_000.LH601_CMD := Rom_000.LH601_CMD;
STLV59_563.STLV59_A_563_000.LH602_CMD := Rom_000.LH602_CMD;
STLV59_563.STLV59_A_563_000.LH603_CMD := Rom_000.LH603_CMD;
STLV59_563.STLV59_A_563_000.LH604_CMD := Rom_000.LH604_CMD;
STLV59_563.STLV59_A_563_000.LH605_CMD := Rom_000.LH605_CMD;
STLV59_563.STLV59_A_563_000.LH606_CMD := Rom_000.LH606_CMD;
STLV59_563.STLV59_A_563_000.LH607_CMD := Rom_000.LH607_CMD;
STLV59_563.STLV59_A_563_000.LH608_CMD := Rom_000.LH608_CMD;
STLV59_563.STLV59_A_563_000.LH609_CMD := Rom_000.LH609_CMD;
STLV59_563.STLV59_A_563_000.LC601_OP := Rom_000.LC601_OP;
STLV59_563.STLV59_A_563_000.LC602_OP := Rom_000.LC602_OP;
STLV59_563.STLV59_A_563_000.LC603_OP := Rom_000.LC603_OP;
STLV59_563.STLV59_A_563_000.LC604_OP := Rom_000.LC604_OP;
STLV59_563.STLV59_A_563_000.LC605_OP := Rom_000.LC605_OP;
STLV59_563.STLV59_A_563_000.LC606_OP := Rom_000.LC606_OP;
STLV59_563.STLV59_A_563_000.LC607_OP := Rom_000.LC607_OP;
STLV59_563.STLV59_A_563_000.LC608_OP := Rom_000.LC608_OP;
STLV59_563.STLV59_A_563_000.LC609_OP := Rom_000.LC609_OP;
STLV59_563.STLV59_A_563_000.LC601_CMD := Rom_000.LC601_CMD;
STLV59_563.STLV59_A_563_000.LC602_CMD := Rom_000.LC602_CMD;
STLV59_563.STLV59_A_563_000.LC603_CMD := Rom_000.LC603_CMD;
STLV59_563.STLV59_A_563_000.LC604_CMD := Rom_000.LC604_CMD;
STLV59_563.STLV59_A_563_000.LC605_CMD := Rom_000.LC605_CMD;
STLV59_563.STLV59_A_563_000.LC606_CMD := Rom_000.LC606_CMD;
STLV59_563.STLV59_A_563_000.LC607_CMD := Rom_000.LC607_CMD;
STLV59_563.STLV59_A_563_000.LC608_CMD := Rom_000.LC608_CMD;
STLV59_563.STLV59_A_563_000.LC609_CMD := Rom_000.LC609_CMD;
STLV59_563.STLV59_A_563_000.LU601_CMD := Rom_000.LU601_CMD;
STLV59_563.STLV59_A_563_000.LU602_CMD := Rom_000.LU602_CMD;
STLV59_563.STLV59_A_563_000.LU603_CMD := Rom_000.LU603_CMD;
STLV59_563.STLV59_A_563_000.LU604_CMD := Rom_000.LU604_CMD;
STLV59_563.STLV59_A_563_000.LU605_CMD := Rom_000.LU605_CMD;
STLV59_563.STLV59_A_563_000.LU606_CMD := Rom_000.LU606_CMD;
STLV59_563.STLV59_A_563_000.LU607_CMD := Rom_000.LU607_CMD;
STLV59_563.STLV59_A_563_000.LU608_CMD := Rom_000.LU608_CMD;
STLV59_563.STLV59_A_563_000.LU609_CMD := Rom_000.LU609_CMD;
(* Rom 001 *)
Rom_001(RB601_HVAC := STLV59_563.STLV59_A_563_001.RB601_HVAC, RB602_HVAC := STLV59_563.STLV59_A_563_001.RB602_HVAC, RT601_CT := STLV59_563.STLV59_A_563_001.RT601_CT, RT601_SP_D := STLV59_563.STLV59_A_563_001.RT601_SP_D, RT601_SP_S := STLV59_563.STLV59_A_563_001.RT601_SP_S, RT601_SP_N := STLV59_563.STLV59_A_563_001.RT601_SP_N, RT601_SP_F := STLV59_563.STLV59_A_563_001.RT601_SP_F, OPM := STLV59_563.STLV59_A_563_001.OPM, LH601_MAN := STLV59_563.STLV59_A_563_001.LH601_MAN, LC601_MAN := STLV59_563.STLV59_A_563_001.LC601_MAN, LU601_V := STLV59_563.STLV59_A_563_001.LU601_V);
STLV59_563.STLV59_A_563_001.OPM_CV := Rom_001.OPM_CV;
STLV59_563.STLV59_A_563_001.RT601_CS := Rom_001.RT601_CS;
STLV59_563.STLV59_A_563_001.LH601_OP := Rom_001.LH601_OP;
STLV59_563.STLV59_A_563_001.LH601_CMD := Rom_001.LH601_CMD;
STLV59_563.STLV59_A_563_001.LC601_OP := Rom_001.LC601_OP;
STLV59_563.STLV59_A_563_001.LC601_CMD := Rom_001.LC601_CMD;
STLV59_563.STLV59_A_563_001.LU601_CMD := Rom_001.LU601_CMD;
(* Rom 002 *)
Rom_002(RB601_HVAC := STLV59_563.STLV59_A_563_002.RB601_HVAC, RT601_CT := STLV59_563.STLV59_A_563_002.RT601_CT, RT602_CT := STLV59_563.STLV59_A_563_002.RT602_CT, RT602_SP := STLV59_563.STLV59_A_563_002.RT602_SP, RT601_SP_D := STLV59_563.STLV59_A_563_002.RT601_SP_D, RT601_SP_S := STLV59_563.STLV59_A_563_002.RT601_SP_S, RT601_SP_N := STLV59_563.STLV59_A_563_002.RT601_SP_N, RT601_SP_F := STLV59_563.STLV59_A_563_002.RT601_SP_F, OPM := STLV59_563.STLV59_A_563_002.OPM, LH601_MAN := STLV59_563.STLV59_A_563_002.LH601_MAN, LC601_MAN := STLV59_563.STLV59_A_563_002.LC601_MAN);
STLV59_563.STLV59_A_563_002.OPM_CV := Rom_002.OPM_CV;
STLV59_563.STLV59_A_563_002.RT601_CS := Rom_002.RT601_CS;
STLV59_563.STLV59_A_563_002.LH601_CMD := Rom_002.LH601_CMD;
STLV59_563.STLV59_A_563_002.LC601_OP := Rom_002.LC601_OP;
(* Rom 004 *)
Rom_004(RB601_HVAC := STLV59_563.STLV59_A_563_004.RB601_HVAC, RT601_CT := STLV59_563.STLV59_A_563_004.RT601_CT, RT602_CT := STLV59_563.STLV59_A_563_004.RT602_CT, RT602_SP := STLV59_563.STLV59_A_563_004.RT602_SP, RT601_SP_D := STLV59_563.STLV59_A_563_004.RT601_SP_D, RT601_SP_S := STLV59_563.STLV59_A_563_004.RT601_SP_S, RT601_SP_N := STLV59_563.STLV59_A_563_004.RT601_SP_N, RT601_SP_F := STLV59_563.STLV59_A_563_004.RT601_SP_F, OPM := STLV59_563.STLV59_A_563_004.OPM, RY601_CV := STLV59_563.STLV59_A_563_004.RY601_CV, RY601_SP := STLV59_563.STLV59_A_563_004.RY601_SP);
STLV59_563.STLV59_A_563_004.OPM_CV := Rom_004.OPM_CV;
STLV59_563.STLV59_A_563_004.RT601_CS := Rom_004.RT601_CS;
STLV59_563.STLV59_A_563_004.RY601_OP := Rom_004.RY601_OP;
(* Rom 005 *)
Rom_005(RB601_HVAC := STLV59_563.STLV59_A_563_005.RB601_HVAC, RT601_CT := STLV59_563.STLV59_A_563_005.RT601_CT, RT602_CT := STLV59_563.STLV59_A_563_005.RT602_CT, RT602_SP := STLV59_563.STLV59_A_563_005.RT602_SP, RT601_SP_D := STLV59_563.STLV59_A_563_005.RT601_SP_D, RT601_SP_S := STLV59_563.STLV59_A_563_005.RT601_SP_S, RT601_SP_N := STLV59_563.STLV59_A_563_005.RT601_SP_N, RT601_SP_F := STLV59_563.STLV59_A_563_005.RT601_SP_F, OPM := STLV59_563.STLV59_A_563_005.OPM, LH601_MAN := STLV59_563.STLV59_A_563_005.LH601_MAN);
STLV59_563.STLV59_A_563_005.OPM_CV := Rom_005.OPM_CV;
STLV59_563.STLV59_A_563_005.RT601_CS := Rom_005.RT601_CS;
STLV59_563.STLV59_A_563_005.LH601_CMD := Rom_005.LH601_CMD;
(* Rom 007 *)
Rom_007(RB601_HVAC := STLV59_563.STLV59_A_563_007.RB601_HVAC, RT601_CT := STLV59_563.STLV59_A_563_007.RT601_CT, RT602_CT := STLV59_563.STLV59_A_563_007.RT602_CT, RT602_SP := STLV59_563.STLV59_A_563_007.RT602_SP, RT601_SP_D := STLV59_563.STLV59_A_563_007.RT601_SP_D, RT601_SP_S := STLV59_563.STLV59_A_563_007.RT601_SP_S, RT601_SP_N := STLV59_563.STLV59_A_563_007.RT601_SP_N, RT601_SP_F := STLV59_563.STLV59_A_563_007.RT601_SP_F, OPM := STLV59_563.STLV59_A_563_007.OPM, LH601_MAN := STLV59_563.STLV59_A_563_007.LH601_MAN);
STLV59_563.STLV59_A_563_007.OPM_CV := Rom_007.OPM_CV;
STLV59_563.STLV59_A_563_007.RT601_CS := Rom_007.RT601_CS;
STLV59_563.STLV59_A_563_007.LH601_CMD := Rom_007.LH601_CMD;
(* Rom 008 *)
Rom_008(RB601_HVAC := STLV59_563.STLV59_A_563_008.RB601_HVAC, RT601_CT := STLV59_563.STLV59_A_563_008.RT601_CT, RT602_CT := STLV59_563.STLV59_A_563_008.RT602_CT, RT602_SP := STLV59_563.STLV59_A_563_008.RT602_SP, RT601_SP_D := STLV59_563.STLV59_A_563_008.RT601_SP_D, RT601_SP_S := STLV59_563.STLV59_A_563_008.RT601_SP_S, RT601_SP_N := STLV59_563.STLV59_A_563_008.RT601_SP_N, RT601_SP_F := STLV59_563.STLV59_A_563_008.RT601_SP_F, OPM := STLV59_563.STLV59_A_563_008.OPM, LH601_MAN := STLV59_563.STLV59_A_563_008.LH601_MAN);
STLV59_563.STLV59_A_563_008.OPM_CV := Rom_008.OPM_CV;
STLV59_563.STLV59_A_563_008.RT601_CS := Rom_008.RT601_CS;
STLV59_563.STLV59_A_563_008.LH601_CMD := Rom_008.LH601_CMD;
(* Rom 009 *)
Rom_009(RB601_HVAC := STLV59_563.STLV59_A_563_009.RB601_HVAC, RT601_CT := STLV59_563.STLV59_A_563_009.RT601_CT, RT602_CT := STLV59_563.STLV59_A_563_009.RT602_CT, RT602_SP := STLV59_563.STLV59_A_563_009.RT602_SP, RT601_SP_D := STLV59_563.STLV59_A_563_009.RT601_SP_D, RT601_SP_S := STLV59_563.STLV59_A_563_009.RT601_SP_S, RT601_SP_N := STLV59_563.STLV59_A_563_009.RT601_SP_N, RT601_SP_F := STLV59_563.STLV59_A_563_009.RT601_SP_F, OPM := STLV59_563.STLV59_A_563_009.OPM, LH601_MAN := STLV59_563.STLV59_A_563_009.LH601_MAN);
STLV59_563.STLV59_A_563_009.OPM_CV := Rom_009.OPM_CV;
STLV59_563.STLV59_A_563_009.RT601_CS := Rom_009.RT601_CS;
STLV59_563.STLV59_A_563_009.LH601_CMD := Rom_009.LH601_CMD;
(* Rom 010 *)
Rom_010(RB601_HVAC := STLV59_563.STLV59_A_563_010.RB601_HVAC, RT601_CT := STLV59_563.STLV59_A_563_010.RT601_CT, RT602_CT := STLV59_563.STLV59_A_563_010.RT602_CT, RT602_SP := STLV59_563.STLV59_A_563_010.RT602_SP, RT601_SP_D := STLV59_563.STLV59_A_563_010.RT601_SP_D, RT601_SP_S := STLV59_563.STLV59_A_563_010.RT601_SP_S, RT601_SP_N := STLV59_563.STLV59_A_563_010.RT601_SP_N, RT601_SP_F := STLV59_563.STLV59_A_563_010.RT601_SP_F, OPM := STLV59_563.STLV59_A_563_010.OPM, LH601_MAN := STLV59_563.STLV59_A_563_010.LH601_MAN);
STLV59_563.STLV59_A_563_010.OPM_CV := Rom_010.OPM_CV;
STLV59_563.STLV59_A_563_010.RT601_CS := Rom_010.RT601_CS;
STLV59_563.STLV59_A_563_010.LH601_CMD := Rom_010.LH601_CMD;
(* Rom 011 *)
Rom_011(RB601_HVAC := STLV59_563.STLV59_A_563_011.RB601_HVAC, RT601_CT := STLV59_563.STLV59_A_563_011.RT601_CT, RT602_CT := STLV59_563.STLV59_A_563_011.RT602_CT, RT602_SP := STLV59_563.STLV59_A_563_011.RT602_SP, RT601_SP_D := STLV59_563.STLV59_A_563_011.RT601_SP_D, RT601_SP_S := STLV59_563.STLV59_A_563_011.RT601_SP_S, RT601_SP_N := STLV59_563.STLV59_A_563_011.RT601_SP_N, RT601_SP_F := STLV59_563.STLV59_A_563_011.RT601_SP_F, OPM := STLV59_563.STLV59_A_563_011.OPM, LH601_MAN := STLV59_563.STLV59_A_563_011.LH601_MAN);
STLV59_563.STLV59_A_563_011.OPM_CV := Rom_011.OPM_CV;
STLV59_563.STLV59_A_563_011.RT601_CS := Rom_011.RT601_CS;
STLV59_563.STLV59_A_563_011.LH601_CMD := Rom_011.LH601_CMD;
(* Rom 012 *)
Rom_012(RB601_HVAC := STLV59_563.STLV59_A_563_012.RB601_HVAC, RT601_CT := STLV59_563.STLV59_A_563_012.RT601_CT, RT602_CT := STLV59_563.STLV59_A_563_012.RT602_CT, RT602_SP := STLV59_563.STLV59_A_563_012.RT602_SP, RT601_SP_D := STLV59_563.STLV59_A_563_012.RT601_SP_D, RT601_SP_S := STLV59_563.STLV59_A_563_012.RT601_SP_S, RT601_SP_N := STLV59_563.STLV59_A_563_012.RT601_SP_N, RT601_SP_F := STLV59_563.STLV59_A_563_012.RT601_SP_F, OPM := STLV59_563.STLV59_A_563_012.OPM, LH601_MAN := STLV59_563.STLV59_A_563_012.LH601_MAN);
STLV59_563.STLV59_A_563_012.OPM_CV := Rom_012.OPM_CV;
STLV59_563.STLV59_A_563_012.RT601_CS := Rom_012.RT601_CS;
STLV59_563.STLV59_A_563_012.LH601_CMD := Rom_012.LH601_CMD;
(* Rom 013 *)
Rom_013(RB601_HVAC := STLV59_563.STLV59_A_563_013.RB601_HVAC, RT601_CT := STLV59_563.STLV59_A_563_013.RT601_CT, RT602_CT := STLV59_563.STLV59_A_563_013.RT602_CT, RT602_SP := STLV59_563.STLV59_A_563_013.RT602_SP, RT601_SP_D := STLV59_563.STLV59_A_563_013.RT601_SP_D, RT601_SP_S := STLV59_563.STLV59_A_563_013.RT601_SP_S, RT601_SP_N := STLV59_563.STLV59_A_563_013.RT601_SP_N, RT601_SP_F := STLV59_563.STLV59_A_563_013.RT601_SP_F, OPM := STLV59_563.STLV59_A_563_013.OPM, LH601_MAN := STLV59_563.STLV59_A_563_013.LH601_MAN);
STLV59_563.STLV59_A_563_013.OPM_CV := Rom_013.OPM_CV;
STLV59_563.STLV59_A_563_013.RT601_CS := Rom_013.RT601_CS;
STLV59_563.STLV59_A_563_013.LH601_CMD := Rom_013.LH601_CMD;
(* Rom 017 *)
Rom_017(RB601_HVAC := STLV59_563.STLV59_A_563_017.RB601_HVAC, RT601_CT := STLV59_563.STLV59_A_563_017.RT601_CT, RT602_CT := STLV59_563.STLV59_A_563_017.RT602_CT, RT602_SP := STLV59_563.STLV59_A_563_017.RT602_SP, RT601_SP_D := STLV59_563.STLV59_A_563_017.RT601_SP_D, RT601_SP_S := STLV59_563.STLV59_A_563_017.RT601_SP_S, RT601_SP_N := STLV59_563.STLV59_A_563_017.RT601_SP_N, RT601_SP_F := STLV59_563.STLV59_A_563_017.RT601_SP_F, OPM := STLV59_563.STLV59_A_563_017.OPM, LH601_MAN := STLV59_563.STLV59_A_563_017.LH601_MAN);
STLV59_563.STLV59_A_563_017.OPM_CV := Rom_017.OPM_CV;
STLV59_563.STLV59_A_563_017.RT601_CS := Rom_017.RT601_CS;
STLV59_563.STLV59_A_563_017.LH601_CMD := Rom_017.LH601_CMD;
(* Rom 101 *)
Rom_101(RB601_HVAC := STLV59_563.STLV59_A_563_101.RB601_HVAC, RT601_CT := STLV59_563.STLV59_A_563_101.RT601_CT, RT602_CT := STLV59_563.STLV59_A_563_101.RT602_CT, RT602_SP := STLV59_563.STLV59_A_563_101.RT602_SP, RT601_SP_D := STLV59_563.STLV59_A_563_101.RT601_SP_D, RT601_SP_S := STLV59_563.STLV59_A_563_101.RT601_SP_S, RT601_SP_N := STLV59_563.STLV59_A_563_101.RT601_SP_N, RT601_SP_F := STLV59_563.STLV59_A_563_101.RT601_SP_F, OPM := STLV59_563.STLV59_A_563_101.OPM, LH601_MAN := STLV59_563.STLV59_A_563_101.LH601_MAN);
STLV59_563.STLV59_A_563_101.OPM_CV := Rom_101.OPM_CV;
STLV59_563.STLV59_A_563_101.RT601_CS := Rom_101.RT601_CS;
STLV59_563.STLV59_A_563_101.LH601_CMD := Rom_101.LH601_CMD;
(* Rom 102 *)
Rom_102(RB601_HVAC := STLV59_563.STLV59_A_563_102.RB601_HVAC, RT601_CT := STLV59_563.STLV59_A_563_102.RT601_CT, RT602_CT := STLV59_563.STLV59_A_563_102.RT602_CT, RT602_SP := STLV59_563.STLV59_A_563_102.RT602_SP, RT601_SP_D := STLV59_563.STLV59_A_563_102.RT601_SP_D, RT601_SP_S := STLV59_563.STLV59_A_563_102.RT601_SP_S, RT601_SP_N := STLV59_563.STLV59_A_563_102.RT601_SP_N, RT601_SP_F := STLV59_563.STLV59_A_563_102.RT601_SP_F, OPM := STLV59_563.STLV59_A_563_102.OPM, LH601_MAN := STLV59_563.STLV59_A_563_102.LH601_MAN);
STLV59_563.STLV59_A_563_102.OPM_CV := Rom_102.OPM_CV;
STLV59_563.STLV59_A_563_102.RT601_CS := Rom_102.RT601_CS;
STLV59_563.STLV59_A_563_102.LH601_CMD := Rom_102.LH601_CMD;
(* Rom 103 *)
Rom_103(RB601_HVAC := STLV59_563.STLV59_A_563_103.RB601_HVAC, RB602_HVAC := STLV59_563.STLV59_A_563_103.RB602_HVAC, RB603_HVAC := STLV59_563.STLV59_A_563_103.RB603_HVAC, RB604_HVAC := STLV59_563.STLV59_A_563_103.RB604_HVAC, RT601_CT := STLV59_563.STLV59_A_563_103.RT601_CT, RT602_CT := STLV59_563.STLV59_A_563_103.RT602_CT, RT602_SP := STLV59_563.STLV59_A_563_103.RT602_SP, RT601_SP_D := STLV59_563.STLV59_A_563_103.RT601_SP_D, RT601_SP_S := STLV59_563.STLV59_A_563_103.RT601_SP_S, RT601_SP_N := STLV59_563.STLV59_A_563_103.RT601_SP_N, RT601_SP_F := STLV59_563.STLV59_A_563_103.RT601_SP_F, OPM := STLV59_563.STLV59_A_563_103.OPM, RY601_CV := STLV59_563.STLV59_A_563_103.RY601_CV, RY601_SP := STLV59_563.STLV59_A_563_103.RY601_SP, LH601_MAN := STLV59_563.STLV59_A_563_103.LH601_MAN, LC601_MAN := STLV59_563.STLV59_A_563_103.LC601_MAN);
STLV59_563.STLV59_A_563_103.OPM_CV := Rom_103.OPM_CV;
STLV59_563.STLV59_A_563_103.RT601_CS := Rom_103.RT601_CS;
STLV59_563.STLV59_A_563_103.RY601_OP := Rom_103.RY601_OP;
STLV59_563.STLV59_A_563_103.LH601_CMD := Rom_103.LH601_CMD;
STLV59_563.STLV59_A_563_103.LC601_OP := Rom_103.LC601_OP;
(* Rom 109 *)
Rom_109(RB601_HVAC := STLV59_563.STLV59_A_563_109.RB601_HVAC, RT601_CT := STLV59_563.STLV59_A_563_109.RT601_CT, RT602_CT := STLV59_563.STLV59_A_563_109.RT602_CT, RT602_SP := STLV59_563.STLV59_A_563_109.RT602_SP, RT601_SP_D := STLV59_563.STLV59_A_563_109.RT601_SP_D, RT601_SP_S := STLV59_563.STLV59_A_563_109.RT601_SP_S, RT601_SP_N := STLV59_563.STLV59_A_563_109.RT601_SP_N, RT601_SP_F := STLV59_563.STLV59_A_563_109.RT601_SP_F, OPM := STLV59_563.STLV59_A_563_109.OPM, LH601_MAN := STLV59_563.STLV59_A_563_109.LH601_MAN);
STLV59_563.STLV59_A_563_109.OPM_CV := Rom_109.OPM_CV;
STLV59_563.STLV59_A_563_109.RT601_CS := Rom_109.RT601_CS;
STLV59_563.STLV59_A_563_109.LH601_CMD := Rom_109.LH601_CMD;
(* Rom 212 *)
Rom_212(RB601_HVAC := STLV59_563.STLV59_A_563_212.RB601_HVAC, RT601_CT := STLV59_563.STLV59_A_563_212.RT601_CT, RT602_CT := STLV59_563.STLV59_A_563_212.RT602_CT, RT602_SP := STLV59_563.STLV59_A_563_212.RT602_SP, RT601_SP_D := STLV59_563.STLV59_A_563_212.RT601_SP_D, RT601_SP_S := STLV59_563.STLV59_A_563_212.RT601_SP_S, RT601_SP_N := STLV59_563.STLV59_A_563_212.RT601_SP_N, RT601_SP_F := STLV59_563.STLV59_A_563_212.RT601_SP_F, OPM := STLV59_563.STLV59_A_563_212.OPM, RY601_CV := STLV59_563.STLV59_A_563_212.RY601_CV, RY601_SP := STLV59_563.STLV59_A_563_212.RY601_SP, LH601_MAN := STLV59_563.STLV59_A_563_212.LH601_MAN, LC601_MAN := STLV59_563.STLV59_A_563_212.LC601_MAN);
STLV59_563.STLV59_A_563_212.OPM_CV := Rom_212.OPM_CV;
STLV59_563.STLV59_A_563_212.RT601_CS := Rom_212.RT601_CS;
STLV59_563.STLV59_A_563_212.RY601_OP := Rom_212.RY601_OP;
STLV59_563.STLV59_A_563_212.LH601_CMD := Rom_212.LH601_CMD;
STLV59_563.STLV59_A_563_212.LC601_OP := Rom_212.LC601_OP;
(* Rom T2_1 *)
Rom_T2_1(RB601_HVAC := STLV59_563.STLV59_A_563_T2_1.RB601_HVAC, RT601_CT := STLV59_563.STLV59_A_563_T2_1.RT601_CT, RT602_CT := STLV59_563.STLV59_A_563_T2_1.RT602_CT, RT602_SP := STLV59_563.STLV59_A_563_T2_1.RT602_SP, RT601_SP_D := STLV59_563.STLV59_A_563_T2_1.RT601_SP_D, RT601_SP_S := STLV59_563.STLV59_A_563_T2_1.RT601_SP_S, RT601_SP_N := STLV59_563.STLV59_A_563_T2_1.RT601_SP_N, RT601_SP_F := STLV59_563.STLV59_A_563_T2_1.RT601_SP_F, OPM := STLV59_563.STLV59_A_563_T2_1.OPM, LH601_MAN := STLV59_563.STLV59_A_563_T2_1.LH601_MAN);
STLV59_563.STLV59_A_563_T2_1.OPM_CV := Rom_T2_1.OPM_CV;
STLV59_563.STLV59_A_563_T2_1.RT601_CS := Rom_T2_1.RT601_CS;
STLV59_563.STLV59_A_563_T2_1.LH601_CMD := Rom_T2_1.LH601_CMD;
(* Rom T2_2 *)
Rom_T2_2(RB601_HVAC := STLV59_563.STLV59_A_563_T2_2.RB601_HVAC, RT601_CT := STLV59_563.STLV59_A_563_T2_2.RT601_CT, RT602_CT := STLV59_563.STLV59_A_563_T2_2.RT602_CT, RT602_SP := STLV59_563.STLV59_A_563_T2_2.RT602_SP, RT601_SP_D := STLV59_563.STLV59_A_563_T2_2.RT601_SP_D, RT601_SP_S := STLV59_563.STLV59_A_563_T2_2.RT601_SP_S, RT601_SP_N := STLV59_563.STLV59_A_563_T2_2.RT601_SP_N, RT601_SP_F := STLV59_563.STLV59_A_563_T2_2.RT601_SP_F, OPM := STLV59_563.STLV59_A_563_T2_2.OPM, LH601_MAN := STLV59_563.STLV59_A_563_T2_2.LH601_MAN);
STLV59_563.STLV59_A_563_T2_2.OPM_CV := Rom_T2_2.OPM_CV;
STLV59_563.STLV59_A_563_T2_2.RT601_CS := Rom_T2_2.RT601_CS;
STLV59_563.STLV59_A_563_T2_2.LH601_CMD := Rom_T2_2.LH601_CMD;
END_PROGRAM
